(* IEC 61131-3 sources: vertical-injection-machine-docs/docs/IM_SYS_PRG/Code/主程序入口, 8 files *)

(* ---- MachineControlTypes.st ---- *)
(*
  MachineControlTypes.st
  功能：
  1. 定义机器级主控入口使用的命令、参数、传感器和状态结构。
  2. 统一手动、调模、半自动、全自动四类运行方式的上层接口。
  3. 为 `FB_MachineController` 和 `PRG_MainControl` 提供稳定的数据边界。

  说明：
  1. 现有各 `FB_*` 子模块仍然保持模块级职责，不在这里重复定义工艺细节。
  2. 机器级接口只负责把分散的模块输入输出汇总成“可实例化、可调用、可监控”的主控层。
  3. 后续若增加新轴、新模块或新工艺模式，应优先扩展本文件，再扩展主控逻辑。
*)

TYPE ST_MachineManualCommand :
STRUCT
    (* 合模模块手动命令。uiClampMode 沿用模块定义：1/2 自动开合模，3/4 调试开合模。 *)
    bClampStart: BOOL;
    uiClampMode: UINT;

    (* 调模模块手动命令。uiMoldAdjustMode 沿用模块定义：1/2 进退，3/4 手动进退。 *)
    bMoldAdjustStart: BOOL;
    uiMoldAdjustMode: UINT;

    (* 座台模块手动命令。uiNozzleMode 沿用模块定义：1/2 进退，3/4 调试进退。 *)
    bNozzleStart: BOOL;
    uiNozzleMode: UINT;

    (* 射胶模块手动命令。uiInjectMode 沿用模块定义：1/2 射出与射退，3/4 调试。 *)
    bInjectStart: BOOL;
    uiInjectMode: UINT;

    (* 储料模块手动命令。储料块没有独立模式号，手动时只需要启动命令。 *)
    bMeterStart: BOOL;

    (* 托模基础模块手动命令。uiEjectMode 沿用模块定义：1/2 进退，6/7 调试。 *)
    bEjectStart: BOOL;
    uiEjectMode: UINT;

    (* 托模组合模式命令。用于定次、震动、停留等更高层动作。 *)
    bEjectModeStart: BOOL;
    uiEjectPatternMode: UINT;   // 1=定次 2=震动 3=停留
    uiEjectTimes: UINT;         // 定次/震动次数；震动模式下 0 表示持续循环

    (* 中子模块手动命令。uiCoreMode 沿用模块定义：1/2 进退，3/4 调试。 *)
    bCoreStart: BOOL;
    uiCoreMode: UINT;

    (* 温控顶层命令。bTempStart 启动温控；bR0~bR3 可直接下发 4 组加热命令。 *)
    bTempStart: BOOL;          // TRUE=顶层温控块进入执行态。
    bR0: BOOL;                 // TRUE=人工直接驱动第 0 组加热输出。
    bR1: BOOL;                 // TRUE=人工直接驱动第 1 组加热输出。
    bR2: BOOL;                 // TRUE=人工直接驱动第 2 组加热输出。
    bR3: BOOL;                 // TRUE=人工直接驱动第 3 组加热输出。
END_STRUCT
END_TYPE

TYPE ST_MachineCommand :
STRUCT
    (* 机器级公共命令。
       说明：
       1. 该结构既可以作为单一命令源边界，也可以作为顶层仲裁后的最终机器命令边界。
       2. 当前工程先接入面板命令源，再由 `FB_CommandArbiter` 统一生成最终 `gvl_stCommand`。
    *)
    bStart: BOOL;               // 周期启动/当前模块启动
    bStop: BOOL;                // 正常停止
    bEStop: BOOL;               // 急停
    bReset: BOOL;               // 复位所有模块

    (* 运行模式。
       0=停机/待机
       1=手动
       2=半自动
       3=全自动
       4=调模模式

       说明：
       1. 手动模式允许人工点动各模块。
       2. 调模模式是独立机器模式，只开放锁模调试与调模相关动作，
          用于装模、试模和模厚调整，不参与自动循环。
    *)
    uiMachineMode: UINT;

    (* 手动模式与调模模式下的分模块命令集合。
       说明：
       1. 手动模式会读取整套人工命令。
       2. 调模模式只会读取其中与锁模调试、调模和温控相关的命令。
    *)
    stManual: ST_MachineManualCommand;
END_STRUCT
END_TYPE

TYPE ST_MachineModeState :
STRUCT
    (* 机器当前模式解析结果。 *)
    bManualModeActive: BOOL;       // TRUE=当前主控解析出的机器模式为手动模式。
    bMoldAdjustModeActive: BOOL;   // TRUE=当前主控解析出的机器模式为调模模式。
    bSemiAutoModeActive: BOOL;     // TRUE=当前主控解析出的机器模式为半自动模式。
    bFullAutoModeActive: BOOL;     // TRUE=当前主控解析出的机器模式为全自动模式。
    bModeChanged: BOOL;            // TRUE=本拍检测到机器模式发生切换，可用于打一拍总停止保护。
    uiResolvedAutoMode: UINT;      // 自动流程专用模式号；0=非自动 1=半自动 2=全自动。
    bGlobalStop: BOOL;             // 主控统一停止位；收口停机命令、停机模式和切模保护停止。
END_STRUCT
END_TYPE

TYPE ST_MachineModuleCommands :
STRUCT
    (* 合模块最终命令。 *)
    bClampStart: BOOL;             // TRUE=主控最终允许合模块启动当前动作。
    bClampReset: BOOL;             // TRUE=主控最终要求合模块回到复位态。
    uiClampMode: UINT;             // 主控最终下发给合模块的动作模式号。

    (* 调模块最终命令。 *)
    bMoldAdjustStart: BOOL;        // TRUE=主控最终允许调模块启动当前动作。
    bMoldAdjustReset: BOOL;        // TRUE=主控最终要求调模块回到复位态。
    uiMoldAdjustMode: UINT;        // 主控最终下发给调模块的动作模式号。

    (* 座台模块最终命令。 *)
    bNozzleStart: BOOL;            // TRUE=主控最终允许座台模块启动当前动作。
    bNozzleReset: BOOL;            // TRUE=主控最终要求座台模块回到复位态。
    uiNozzleMode: UINT;            // 主控最终下发给座台模块的动作模式号。

    (* 射胶模块最终命令。 *)
    bInjectStart: BOOL;            // TRUE=主控最终允许射胶模块启动当前动作。
    bInjectReset: BOOL;            // TRUE=主控最终要求射胶模块回到复位态。
    uiInjectMode: UINT;            // 主控最终下发给射胶模块的动作模式号。

    (* 储料模块最终命令。 *)
    bMeterStart: BOOL;             // TRUE=主控最终允许储料模块启动当前动作。
    bMeterReset: BOOL;             // TRUE=主控最终要求储料模块回到复位态。

    (* 基础托模块最终命令。 *)
    bEjectStart: BOOL;             // TRUE=主控最终允许基础托模块启动当前动作。
    bEjectReset: BOOL;             // TRUE=主控最终要求基础托模块回到复位态。
    uiEjectMode: UINT;             // 主控最终下发给基础托模块的动作模式号。

    (* 托模组合模式块最终命令。 *)
    bEjectModeStart: BOOL;         // TRUE=主控最终允许托模组合模式块启动当前动作。
    bEjectModeReset: BOOL;         // TRUE=主控最终要求托模组合模式块回到复位态。
    uiEjectPatternMode: UINT;      // 主控最终下发给托模组合模式块的组合模式号。
    uiEjectTimes: UINT;            // 主控最终下发给托模组合模式块的循环次数或震动次数。

    (* 中子模块最终命令。 *)
    bCoreStart: BOOL;              // TRUE=主控最终允许中子模块启动当前动作。
    bCoreReset: BOOL;              // TRUE=主控最终要求中子模块回到复位态。
    uiCoreMode: UINT;              // 主控最终下发给中子模块的动作模式号。
END_STRUCT
END_TYPE

TYPE ST_MachineSensor :
STRUCT
    (* 机器公共条件。自动流程会优先检查这些前提是否满足。 *)
    bDoorClosed: BOOL;
    bHydReady: BOOL;
    bSystemNoAlarm: BOOL;

    (* 合模模块过程信号。 *)
    bOpenStop: BOOL;
    bCloseLowPres: BOOL;
    bCloseHighPres: BOOL;
    bCloseStop: BOOL;
    udiClampElecRulerVal: UDINT;
    uiClampPresElecRulerVal: UINT;

    (* 调模模块过程信号。 *)
    bMoldAdjustInStop: BOOL;
    bMoldAdjustOutStop: BOOL;

    (* 座台模块过程信号。 *)
    bNozzleInStop: BOOL;
    bNozzleOutStop: BOOL;
    udiNozzleElecRulerVal: UDINT;

    (* 射胶与储料模块过程信号。 *)
    bInjSeg1Stop: BOOL;
    bInjSeg2Stop: BOOL;
    bInjStop: BOOL;
    bSuckBackStop: BOOL;
    bMeterStop: BOOL;
    udiInjElecRulerVal: UDINT;

    (* 托模模块过程信号。 *)
    bEjectInStop: BOOL;
    bEjectOutStop: BOOL;
    udiEjectElecRulerVal: UDINT;

    (* 中子模块过程信号。 *)
    bCoreInStop: BOOL;
    bCoreOutStop: BOOL;

    (* 轴反馈。
       这些反馈值会经由子模块接口写回各自的 `ST_AxisRefHyd`，让模块层同时看到“设定值”和“实际值”。
    *)
    rClampActualPosition: LREAL;
    rClampActualVelocity: LREAL;
    rClampActualPressure: LREAL;

    rMoldAdjustActualPosition: LREAL;
    rMoldAdjustActualVelocity: LREAL;
    rMoldAdjustActualPressure: LREAL;

    rNozzleActualPosition: LREAL;
    rNozzleActualVelocity: LREAL;
    rNozzleActualPressure: LREAL;

    rInjectActualPosition: LREAL;
    rInjectActualVelocity: LREAL;
    rInjectActualPressure: LREAL;

    rMeterActualPosition: LREAL;
    rMeterActualVelocity: LREAL;
    rMeterActualPressure: LREAL;

    rEjectActualPosition: LREAL;
    rEjectActualVelocity: LREAL;
    rEjectActualPressure: LREAL;

    rCoreActualPosition: LREAL;
    rCoreActualVelocity: LREAL;
    rCoreActualPressure: LREAL;
END_STRUCT
END_TYPE

TYPE ST_MachinePara :
STRUCT
    (* 子模块工艺参数全集。
       说明：
       1. 这是机器当前在线运行参数。
       2. `FB_MachineController` 只读取并分发，不在内部改写这些工艺值。
       3. 若 HMI 需要统一配方编辑入口，建议通过专用 HMI 参数接口先写入编辑缓冲区，
          再由上层执行“应用到机器”动作，避免画面直接改动在线参数。
    *)
    stClampPara: ST_ClampPara;
    stMoldAdjustPara: ST_MoldAdjustPara;
    stNozzlePara: ST_NozzlePara;
    stInjectPara: ST_InjectPara;
    stMeterPara: ST_MeterPara;
    stEjectPara: ST_EjectPara;
    stCorePara: ST_CorePara;
    stEK312InPara: ST_EK312InPara;
    stAutoPara: ST_AutoCyclePara;
END_STRUCT
END_TYPE

TYPE ST_HMIRecipeMeta :
STRUCT
    (* HMI 配方基础信息。
       这些字段不直接参与动作控制，但便于画面做配方编号、名称、版本和脏数据管理。
    *)
    uiRecipeID: UINT;             // HMI 配方号/工艺号
    sRecipeName: STRING[40];      // HMI 显示用配方名称
    uiRecipeVersion: UINT;        // HMI 自管版本号，可在每次保存后自增
    bDirty: BOOL;                 // TRUE=HMI 编辑缓冲区已改动但还未下发到机器
END_STRUCT
END_TYPE

TYPE ST_HMIProcessPara :
STRUCT
    (* HMI 统一工艺参数接口。
       说明：
       1. HMI 只需要绑定这一套结构，就能覆盖整机全部工艺参数。
       2. 内部仍复用各模块原生参数结构，避免为了画面再拆一层重复字段。
       3. `stMachinePara` 是 HMI 编辑缓冲区，不等同于当前在线运行参数。
          只有执行“应用到机器”后，内容才会写入在线参数。
       4. HMI 画面在用户改动任意字段后，建议同步把 `stMeta.bDirty` 置为 TRUE，
          便于配方页显示“已编辑未下发/未保存”状态。
    *)
    stMeta: ST_HMIRecipeMeta;
    stMachinePara: ST_MachinePara;
END_STRUCT
END_TYPE

TYPE ST_HMIParaCommand :
STRUCT
    (* HMI 参数同步命令。
       这些信号建议由按钮上升沿触发，不建议长时间保持 TRUE。
    *)
    bReadMachinePara: BOOL;       // 把当前在线运行参数读回到 HMI 编辑缓冲区
    bApplyToMachine: BOOL;        // 把 HMI 编辑缓冲区参数应用到机器在线参数
    bClearDirty: BOOL;            // 人工清除 HMI 编辑脏标记
END_STRUCT
END_TYPE

TYPE ST_HMIParaStatus :
STRUCT
    (* HMI 参数接口状态。
       这些状态用于给 HMI 做按钮反馈、提示灯和下发拦截提示。
    *)
    bInitialized: BOOL;           // TRUE=已完成首次把在线参数装载到 HMI 缓冲区
    bMachineParaLocked: BOOL;     // TRUE=机器正在运行/忙碌，禁止下发工艺参数
    bReadDone: BOOL;              // 本扫描周期完成了一次在线参数读回
    bApplyDone: BOOL;             // 本扫描周期完成了一次工艺参数下发
    bClearDone: BOOL;             // 本扫描周期完成了一次脏标记清除
    bApplyBlocked: BOOL;          // 本扫描周期收到下发命令但被拦截
    uiLastAction: UINT;           // 0=无 1=首次装载 2=读取在线参数 3=应用到机器 4=清除脏标记 5=下发被拦截
    uiLastRejectReason: UINT;     // 0=无 1=机器忙碌
    uiSyncCount: UINT;            // 成功同步次数统计
    uiRecipeID: UINT;             // 当前 HMI 缓冲区配方号镜像
    uiRecipeVersion: UINT;        // 当前 HMI 缓冲区版本号镜像
    sRecipeName: STRING[40];      // 当前 HMI 缓冲区名称镜像
    bDirty: BOOL;                 // 当前 HMI 缓冲区脏标记镜像
END_STRUCT
END_TYPE

TYPE ST_MachineStatus :
STRUCT
    (* 机器级总状态。 *)
    uiMachineMode: UINT;
    bManualModeActive: BOOL;
    bMoldAdjustModeActive: BOOL;
    bSemiAutoModeActive: BOOL;
    bFullAutoModeActive: BOOL;
    bAutoReady: BOOL;
    bMachineBusy: BOOL;
    bMachineDone: BOOL;
    bMachineAlarm: BOOL;
    dwMachineAlarmID: DWORD;
    uiMachineActHint: UINT;
    uiMachineActTime: UINT;
    uiCycleCount: UINT;

    (* 自动流程状态。 *)
    bAutoBusy: BOOL;
    bAutoDone: BOOL;
    bAutoAlarm: BOOL;
    dwAutoAlarmID: DWORD;

    (* 合模模块状态。 *)
    bClampBusy: BOOL;
    bClampDone: BOOL;
    bClampAlarm: BOOL;
    dwClampAlarmID: DWORD;
    bMoldOpened: BOOL;
    bMoldClosed: BOOL;

    (* 调模模块状态。 *)
    bMoldAdjustBusy: BOOL;
    bMoldAdjustDone: BOOL;
    bMoldAdjustAlarm: BOOL;
    dwMoldAdjustAlarmID: DWORD;
    bMoldAdjustIned: BOOL;
    bMoldAdjustOuted: BOOL;

    (* 座台模块状态。 *)
    bNozzleBusy: BOOL;
    bNozzleDone: BOOL;
    bNozzleAlarm: BOOL;
    dwNozzleAlarmID: DWORD;
    bNozzleIned: BOOL;
    bNozzleOuted: BOOL;

    (* 射胶模块状态。 *)
    bInjectBusy: BOOL;
    bInjectDone: BOOL;
    bInjectAlarm: BOOL;
    dwInjectAlarmID: DWORD;
    bInjected: BOOL;
    bHeld: BOOL;
    bSuckBacked: BOOL;

    (* 储料模块状态。 *)
    bMeterBusy: BOOL;
    bMeterDone: BOOL;
    bMeterAlarm: BOOL;
    dwMeterAlarmID: DWORD;
    bMetered: BOOL;

    (* 托模模块状态。
       bEjectModeSelected=TRUE 时表示当前输出来自 `FB_EjectMode`；
       否则当前输出来自基础 `FB_Eject`。
    *)
    bEjectModeSelected: BOOL;
    bEjectBusy: BOOL;
    bEjectDone: BOOL;
    bEjectAlarm: BOOL;
    dwEjectAlarmID: DWORD;
    bEjectIned: BOOL;
    bEjectOuted: BOOL;

    (* 中子模块状态。 *)
    bCoreBusy: BOOL;
    bCoreDone: BOOL;
    bCoreAlarm: BOOL;
    dwCoreAlarmID: DWORD;
    bCoreIned: BOOL;
    bCoreOuted: BOOL;

END_STRUCT
END_TYPE

(* ---- FB_CommandArbiter.st ---- *)
(*
  FB_CommandArbiter 功能块
  功能：
  1. 统一收口顶层不同来源的机器命令，再输出给 `FB_MachineController` 与其他顶层消费者。
  2. 当前版本先保留外部入口已经写入的基础公共命令，再用面板命令源覆盖模式与手动字段。
  3. 后续若接入 HMI 运行命令、远程命令或调试命令，应优先在本块扩展优先级与仲裁规则。
*)
FUNCTION_BLOCK FB_CommandArbiter
VAR_INPUT
    stBaseCommandIn: ST_MachineCommand;          // 其他外部入口当前写入的基础机器命令快照；当前版本优先保留其公共启动/停止/复位类字段。
    stPanelCommandSourceIn: ST_MachineCommand;   // 面板调度层输出的机器命令源；当前版本只用本源覆盖模式与手动字段，不直接覆盖公共启动/停止/复位类字段。
END_VAR
VAR_OUTPUT
    stCommandOut: ST_MachineCommand;             // 仲裁后的最终机器命令；供顶层温控和机器主控统一消费。
END_VAR

(* 当前版本的仲裁策略：
   1. 先保留外部基础命令快照中的公共启动/停止/复位/EStop 字段。
   2. 再用面板命令源覆盖它真正负责的模式与手动点动字段。
   3. 这里保留独立功能块，是为了后续增加新命令源时不再修改顶层调用链。
*)
stCommandOut := stBaseCommandIn;                                               // 先复制当前扫描周期的基础机器命令快照，保留外部入口写入的公共控制字段。

IF stPanelCommandSourceIn.uiMachineMode <> UINT#0 THEN
    stCommandOut.uiMachineMode := stPanelCommandSourceIn.uiMachineMode;         // 面板只要给出了有效模式号，就由面板模式选择覆盖当前最终机器模式。
END_IF;

stCommandOut.stManual.bClampStart := stPanelCommandSourceIn.stManual.bClampStart;                 // 合模点动命令由面板源直接覆盖最终手动命令。
stCommandOut.stManual.uiClampMode := stPanelCommandSourceIn.stManual.uiClampMode;                 // 合模点动模式号由面板源直接覆盖最终手动命令。
stCommandOut.stManual.bMoldAdjustStart := stPanelCommandSourceIn.stManual.bMoldAdjustStart;       // 调模点动命令由面板源直接覆盖最终手动命令。
stCommandOut.stManual.uiMoldAdjustMode := stPanelCommandSourceIn.stManual.uiMoldAdjustMode;       // 调模点动模式号由面板源直接覆盖最终手动命令。
stCommandOut.stManual.bNozzleStart := stPanelCommandSourceIn.stManual.bNozzleStart;               // 座台点动命令由面板源直接覆盖最终手动命令。
stCommandOut.stManual.uiNozzleMode := stPanelCommandSourceIn.stManual.uiNozzleMode;               // 座台点动模式号由面板源直接覆盖最终手动命令。
stCommandOut.stManual.bInjectStart := stPanelCommandSourceIn.stManual.bInjectStart;               // 射胶点动命令由面板源直接覆盖最终手动命令。
stCommandOut.stManual.uiInjectMode := stPanelCommandSourceIn.stManual.uiInjectMode;               // 射胶点动模式号由面板源直接覆盖最终手动命令。
stCommandOut.stManual.bMeterStart := stPanelCommandSourceIn.stManual.bMeterStart;                 // 储料点动命令由面板源直接覆盖最终手动命令。
stCommandOut.stManual.bEjectStart := stPanelCommandSourceIn.stManual.bEjectStart;                 // 基础托模点动命令由面板源直接覆盖最终手动命令。
stCommandOut.stManual.uiEjectMode := stPanelCommandSourceIn.stManual.uiEjectMode;                 // 基础托模模式号由面板源直接覆盖最终手动命令。
stCommandOut.stManual.bEjectModeStart := stPanelCommandSourceIn.stManual.bEjectModeStart;         // 托模组合模式启动命令由面板源直接覆盖最终手动命令。
stCommandOut.stManual.uiEjectPatternMode := stPanelCommandSourceIn.stManual.uiEjectPatternMode;   // 托模组合模式号由面板源直接覆盖最终手动命令。
stCommandOut.stManual.uiEjectTimes := stPanelCommandSourceIn.stManual.uiEjectTimes;               // 托模组合次数由面板源直接覆盖最终手动命令。
stCommandOut.stManual.bCoreStart := stPanelCommandSourceIn.stManual.bCoreStart;                   // 中子点动命令由面板源直接覆盖最终手动命令。
stCommandOut.stManual.uiCoreMode := stPanelCommandSourceIn.stManual.uiCoreMode;                   // 中子点动模式号由面板源直接覆盖最终手动命令。
stCommandOut.stManual.bTempStart := stPanelCommandSourceIn.stManual.bTempStart;                   // 温控开关锁存值由面板源直接覆盖最终手动命令。
stCommandOut.stManual.bR0 := stPanelCommandSourceIn.stManual.bR0;                                 // 温控人工组 0 命令由面板源直接覆盖最终手动命令。
stCommandOut.stManual.bR1 := stPanelCommandSourceIn.stManual.bR1;                                 // 温控人工组 1 命令由面板源直接覆盖最终手动命令。
stCommandOut.stManual.bR2 := stPanelCommandSourceIn.stManual.bR2;                                 // 温控人工组 2 命令由面板源直接覆盖最终手动命令。
stCommandOut.stManual.bR3 := stPanelCommandSourceIn.stManual.bR3;                                 // 温控人工组 3 命令由面板源直接覆盖最终手动命令。
END_FUNCTION_BLOCK

(* ---- FB_MachineCommandComposer.st ---- *)
(*
  FB_MachineCommandComposer 功能块
  功能：
  1. 把手动、调模和自动三类来源的模块命令合成为一套最终执行命令。
  2. 把基础托模块与托模组合模式块的互斥选择统一收口，避免双块抢同一根轴。
  3. 当前块只负责命令合成，不直接调用任何执行模块。
*)
FUNCTION_BLOCK FB_MachineCommandComposer
VAR_INPUT
    stCommand: ST_MachineCommand;            // 顶层下发的最终机器命令；当前块只消费公共复位命令与手动命令结构。
    stModeState: ST_MachineModeState;        // 当前扫描周期解析出的模式状态结构；决定最终命令应由哪一类来源接管。

    (* 手动/调模路由结果。 *)
    bManualClampStart: BOOL;                 // 手动或调模路由给出的合模启动命令。
    uiManualClampMode: UINT;                 // 手动或调模路由给出的合模模式号。
    bManualMoldAdjustStart: BOOL;            // 手动或调模路由给出的调模启动命令。
    uiManualMoldAdjustMode: UINT;            // 手动或调模路由给出的调模模式号。
    bManualNozzleStart: BOOL;                // 手动路由给出的座台启动命令。
    uiManualNozzleMode: UINT;                // 手动路由给出的座台模式号。
    bManualInjectStart: BOOL;                // 手动路由给出的射胶启动命令。
    uiManualInjectMode: UINT;                // 手动路由给出的射胶模式号。
    bManualMeterStart: BOOL;                 // 手动路由给出的储料启动命令。
    bManualEjectStart: BOOL;                 // 手动路由给出的基础托模启动命令。
    uiManualEjectMode: UINT;                 // 手动路由给出的基础托模模式号。
    bManualEjectModeStart: BOOL;             // 手动路由给出的托模组合模式启动命令。
    uiManualEjectPatternMode: UINT;          // 手动路由给出的托模组合模式号。
    uiManualEjectTimes: UINT;                // 手动路由给出的托模组合次数或震动次数。
    bManualCoreStart: BOOL;                  // 手动路由给出的中子启动命令。
    uiManualCoreMode: UINT;                  // 手动路由给出的中子模式号。

    (* 自动流程输出结果。 *)
    bAutoClampStart: BOOL;                   // 自动流程给出的合模启动命令。
    bAutoClampReset: BOOL;                   // 自动流程给出的合模复位命令。
    uiAutoClampMode: UINT;                   // 自动流程给出的合模模式号。
    bAutoNozzleStart: BOOL;                  // 自动流程给出的座台启动命令。
    bAutoNozzleReset: BOOL;                  // 自动流程给出的座台复位命令。
    uiAutoNozzleMode: UINT;                  // 自动流程给出的座台模式号。
    bAutoInjectStart: BOOL;                  // 自动流程给出的射胶启动命令。
    bAutoInjectReset: BOOL;                  // 自动流程给出的射胶复位命令。
    uiAutoInjectMode: UINT;                  // 自动流程给出的射胶模式号。
    bAutoMeterStart: BOOL;                   // 自动流程给出的储料启动命令。
    bAutoMeterReset: BOOL;                   // 自动流程给出的储料复位命令。
    bAutoEjectStart: BOOL;                   // 自动流程给出的基础托模启动命令。
    bAutoEjectReset: BOOL;                   // 自动流程给出的基础托模复位命令。
    uiAutoEjectMode: UINT;                   // 自动流程给出的基础托模模式号。
END_VAR
VAR_OUTPUT
    stModuleCommands: ST_MachineModuleCommands; // 主控最终下发给各执行模块的统一命令集合。
    bUseEjectModeManual: BOOL;                  // TRUE=当前应切换到托模组合模式块，而不是基础托模块。
END_VAR

(* 先给各模块命令做安全缺省值。
   这样在模式切换时，未被当前模式接管的模块会自然保持停止/复位，不会沿用旧命令。
*)
stModuleCommands.bClampStart := FALSE;                          // 默认不给合模块启动命令，避免未被接管时沿用旧动作。
stModuleCommands.bClampReset := stCommand.bReset;              // 合模块默认只响应顶层复位命令。
stModuleCommands.uiClampMode := 0;                             // 合模块默认模式号清零，表示当前无有效动作。

stModuleCommands.bMoldAdjustStart := FALSE;                    // 默认不给调模块启动命令，避免未被接管时沿用旧动作。
stModuleCommands.bMoldAdjustReset := stCommand.bReset;         // 调模块默认只响应顶层复位命令。
stModuleCommands.uiMoldAdjustMode := 0;                        // 调模块默认模式号清零，表示当前无有效动作。

stModuleCommands.bNozzleStart := FALSE;                        // 默认不给座台模块启动命令，避免未被接管时沿用旧动作。
stModuleCommands.bNozzleReset := stCommand.bReset;             // 座台模块默认只响应顶层复位命令。
stModuleCommands.uiNozzleMode := 0;                            // 座台模块默认模式号清零，表示当前无有效动作。

stModuleCommands.bInjectStart := FALSE;                        // 默认不给射胶模块启动命令，避免未被接管时沿用旧动作。
stModuleCommands.bInjectReset := stCommand.bReset;             // 射胶模块默认只响应顶层复位命令。
stModuleCommands.uiInjectMode := 0;                            // 射胶模块默认模式号清零，表示当前无有效动作。

stModuleCommands.bMeterStart := FALSE;                         // 默认不给储料模块启动命令，避免未被接管时沿用旧动作。
stModuleCommands.bMeterReset := stCommand.bReset;              // 储料模块默认只响应顶层复位命令。

stModuleCommands.bEjectStart := FALSE;                         // 默认不给基础托模块启动命令，避免未被接管时沿用旧动作。
stModuleCommands.bEjectReset := stCommand.bReset;              // 基础托模块默认只响应顶层复位命令。
stModuleCommands.uiEjectMode := 0;                             // 基础托模块默认模式号清零，表示当前无有效动作。

stModuleCommands.bEjectModeStart := FALSE;                     // 默认不给托模模式块启动命令，避免组合模式在切模后残留。
stModuleCommands.bEjectModeReset := TRUE;                      // 默认把托模模式块拉在复位态，只有明确使用时才释放。
stModuleCommands.uiEjectPatternMode := 0;                      // 托模模式块默认模式号清零，表示当前不执行组合动作。
stModuleCommands.uiEjectTimes := 0;                            // 托模模式块默认次数清零，避免沿用上一轮次数设定。

stModuleCommands.bCoreStart := FALSE;                          // 默认不给中子模块启动命令，避免未被接管时沿用旧动作。
stModuleCommands.bCoreReset := stCommand.bReset;               // 中子模块默认只响应顶层复位命令。
stModuleCommands.uiCoreMode := 0;                              // 中子模块默认模式号清零，表示当前无有效动作。

(* 把不同来源的命令合并为“最终执行命令”。
   1. 手动模式：手动命令由 `FB_ManualMode` 路由。
   2. 调模模式：命令由 `FB_MoldAdjustMode` 路由，锁模强制进入调试方向，其他模块保持停机。
   3. 自动模式：命令来自 `FB_AutoCycle` 的调度输出。
*)
IF stModeState.bManualModeActive THEN
    stModuleCommands.bClampStart := bManualClampStart;             // 手动模式下，合模块直接接收手动命令路由结果。
    stModuleCommands.uiClampMode := uiManualClampMode;             // 手动模式下，合模块直接接收手动动作模式号。

    stModuleCommands.bMoldAdjustStart := bManualMoldAdjustStart;   // 手动模式下，调模块直接接收手动命令路由结果。
    stModuleCommands.uiMoldAdjustMode := uiManualMoldAdjustMode;   // 手动模式下，调模块直接接收手动动作模式号。

    stModuleCommands.bNozzleStart := bManualNozzleStart;           // 手动模式下，座台模块直接接收手动命令路由结果。
    stModuleCommands.uiNozzleMode := uiManualNozzleMode;           // 手动模式下，座台模块直接接收手动动作模式号。

    stModuleCommands.bInjectStart := bManualInjectStart;           // 手动模式下，射胶模块直接接收手动命令路由结果。
    stModuleCommands.uiInjectMode := uiManualInjectMode;           // 手动模式下，射胶模块直接接收手动动作模式号。

    stModuleCommands.bMeterStart := bManualMeterStart;             // 手动模式下，储料模块直接接收手动启动命令。

    stModuleCommands.bCoreStart := bManualCoreStart;               // 手动模式下，中子模块直接接收手动命令路由结果。
    stModuleCommands.uiCoreMode := uiManualCoreMode;               // 手动模式下，中子模块直接接收手动动作模式号。
ELSIF stModeState.bMoldAdjustModeActive THEN
    stModuleCommands.bClampStart := bManualClampStart;             // 调模模式下，锁模动作仍由调模命令路由结果接管。
    stModuleCommands.uiClampMode := uiManualClampMode;             // 调模模式下，锁模模式号仍取自调模命令路由结果。

    stModuleCommands.bMoldAdjustStart := bManualMoldAdjustStart;   // 调模模式下，调模块直接接收调模命令路由结果。
    stModuleCommands.uiMoldAdjustMode := uiManualMoldAdjustMode;   // 调模模式下，调模块直接接收调模动作模式号。
ELSE
    stModuleCommands.bClampStart := bAutoClampStart;               // 自动模式下，合模块启动命令由自动流程输出接管。
    stModuleCommands.bClampReset := stCommand.bReset OR bAutoClampReset; // 自动模式下，顶层复位与自动步骤复位任一成立都可复位合模块。
    stModuleCommands.uiClampMode := uiAutoClampMode;               // 自动模式下，合模块动作模式号由自动流程给定。

    stModuleCommands.bNozzleStart := bAutoNozzleStart;             // 自动模式下，座台模块启动命令由自动流程输出接管。
    stModuleCommands.bNozzleReset := stCommand.bReset OR bAutoNozzleReset; // 自动模式下，顶层复位与自动步骤复位任一成立都可复位座台模块。
    stModuleCommands.uiNozzleMode := uiAutoNozzleMode;             // 自动模式下，座台模块动作模式号由自动流程给定。

    stModuleCommands.bInjectStart := bAutoInjectStart;             // 自动模式下，射胶模块启动命令由自动流程输出接管。
    stModuleCommands.bInjectReset := stCommand.bReset OR bAutoInjectReset; // 自动模式下，顶层复位与自动步骤复位任一成立都可复位射胶模块。
    stModuleCommands.uiInjectMode := uiAutoInjectMode;             // 自动模式下，射胶模块动作模式号由自动流程给定。

    stModuleCommands.bMeterStart := bAutoMeterStart;               // 自动模式下，储料模块启动命令由自动流程输出接管。
    stModuleCommands.bMeterReset := stCommand.bReset OR bAutoMeterReset; // 自动模式下，顶层复位与自动步骤复位任一成立都可复位储料模块。

    stModuleCommands.bEjectStart := bAutoEjectStart;               // 自动模式下，基础托模块启动命令由自动流程输出接管。
    stModuleCommands.bEjectReset := stCommand.bReset OR bAutoEjectReset; // 自动模式下，顶层复位与自动步骤复位任一成立都可复位基础托模块。
    stModuleCommands.uiEjectMode := uiAutoEjectMode;               // 自动模式下，基础托模块动作模式号由自动流程给定。
END_IF;

(* 托模既有基础动作块，也有组合模式块。
   这里把两类命令拆开，避免两个功能块同时争抢同一输出轴。
*)
bUseEjectModeManual := stModeState.bManualModeActive AND bManualEjectModeStart AND   // 只有手动模式下明确发起托模模式命令时，才允许切到组合托模块。
    (uiManualEjectPatternMode >= 1) AND                                               // 模式号下限必须落在当前支持的托模组合模式范围内。
    (uiManualEjectPatternMode <= 3);                                                  // 模式号上限必须落在当前支持的托模组合模式范围内。

IF stModeState.bManualModeActive AND (NOT bUseEjectModeManual) THEN
    stModuleCommands.bEjectStart := bManualEjectStart;               // 纯手动基础托模时，把基础托模启动命令路由给 `FB_Eject`。
    stModuleCommands.bEjectReset := stCommand.bReset;                // 纯手动基础托模时，基础托模块只响应顶层复位命令。
    stModuleCommands.uiEjectMode := uiManualEjectMode;               // 纯手动基础托模时，把手动托模模式号路由给 `FB_Eject`。
ELSIF NOT stModeState.bManualModeActive THEN
    stModuleCommands.bEjectStart := bAutoEjectStart;                 // 非手动模式下，基础托模块启动命令由自动流程输出接管。
    stModuleCommands.bEjectReset := stCommand.bReset OR bAutoEjectReset; // 非手动模式下，顶层复位与自动步骤复位任一成立都可复位基础托模块。
    stModuleCommands.uiEjectMode := uiAutoEjectMode;                 // 非手动模式下，基础托模块动作模式号由自动流程给定。
ELSE
    stModuleCommands.bEjectStart := FALSE;                           // 进入托模组合模式时，强制撤销基础托模块启动命令，避免双块抢轴。
    stModuleCommands.bEjectReset := TRUE;                            // 进入托模组合模式时，强制把基础托模块拉回复位态。
    stModuleCommands.uiEjectMode := 0;                               // 进入托模组合模式时，基础托模块模式号清零。
END_IF;

IF bUseEjectModeManual THEN
    stModuleCommands.bEjectModeStart := bManualEjectModeStart;       // 仅在手动组合托模生效时，把启动命令路由给 `FB_EjectMode`。
    stModuleCommands.bEjectModeReset := stCommand.bReset;            // 仅在手动组合托模生效时，把顶层复位命令路由给 `FB_EjectMode`。
    stModuleCommands.uiEjectPatternMode := uiManualEjectPatternMode; // 仅在手动组合托模生效时，把托模组合模式号路由给 `FB_EjectMode`。
    stModuleCommands.uiEjectTimes := uiManualEjectTimes;             // 仅在手动组合托模生效时，把循环次数或震动次数路由给 `FB_EjectMode`。
END_IF;
END_FUNCTION_BLOCK

(* ---- FB_MachineController.st ---- *)
(*
  FB_MachineController 功能块
  功能：
  1. 提供真正的机器级执行层，负责实例化并周期调用所有模块级功能块。
  2. 通过内部辅助层完成模式解析、命令合成，并把最终模块命令分发给各执行块。
  3. 把模块状态、轴命令和自动流程状态汇总为统一的机器级状态输出。

  调用关系：
  1. `FB_MachineModeResolver` 只负责模式解析，不直接驱动任何执行模块。
  2. `FB_AutoCycle` 只负责调度，不直接驱动任何轴；`FB_MachineCommandComposer` 负责把自动、手动和调模命令收口为最终模块命令。
  3. 各执行模块内部各自持有 `FB_HydAxis` 并自行处理轴使能、轴配置和轴状态并入。
  4. `FB_MachineStatusAggregator` 负责把自动流程和模块状态收口为机器总状态。
  5. `FB_EK312` 由 `PROGRAM PRG_MainControl` 顶层独立调用，本功能块不处理温控块接口和温控状态。
  6. 必须由 `PROGRAM PRG_MainControl` 以 1ms 基础任务调用本功能块；10ms 工艺节拍也必须由顶层生成后通过输入接口送入本块。
*)
FUNCTION_BLOCK FB_MachineController
VAR_INPUT
    stCommand: ST_MachineCommand;    // 顶层下发的机器公共命令集合，包含启动/停止/复位/模式号以及手动动作命令。
    stPara: ST_MachinePara;          // 顶层下发的机器在线工艺参数全集，由主控分发给各执行模块使用。
    stSensor: ST_MachineSensor;      // 顶层采集的现场条件、限位和轴反馈，供主控与子模块做互锁和状态判断。
    bLogicTick10msIn: BOOL;          // 顶层当前扫描周期给出的 10ms 工艺逻辑节拍，本块只在该拍刷新模式路由和自动流程。
END_VAR
VAR_OUTPUT
    stStatus: ST_MachineStatus;      // 主控汇总后的机器级总状态，供 HMI、上位机和其他顶层逻辑统一读取。

    (* 各轴输出。
       这些结构体同时包含模块下发的设定值与主控层回写的实际反馈值，
       便于后续继续接入真实轴控或液压阀控层。
    *)
    stClampAxis: ST_AxisRefHyd;          // 合模模块输出的最终轴命令与反馈镜像，对外暴露为锁模轴边界。
    stMoldAdjustAxis: ST_AxisRefHyd;     // 调模模块输出的最终轴命令与反馈镜像，对外暴露为调模轴边界。
    stNozzleAxis: ST_AxisRefHyd;         // 座台模块输出的最终轴命令与反馈镜像，对外暴露为座台轴边界。
    stInjectAxis: ST_AxisRefHyd;         // 射胶模块输出的最终轴命令与反馈镜像，对外暴露为射胶轴边界。
    stMeterAxis: ST_AxisRefHyd;          // 储料模块输出的最终轴命令与反馈镜像，对外暴露为储料轴边界。
    stEjectAxis: ST_AxisRefHyd;          // 托模模块当前被选中的最终轴命令与反馈镜像，可能来自基础托模或托模模式。
    stCoreAxis: ST_AxisRefHyd;           // 中子模块输出的最终轴命令与反馈镜像，对外暴露为中子轴边界。

    (* 透传关键组合输出。 *)
    aCoreAllow: ARRAY[1..8] OF BOOL;     // 合模模块回写的 8 路中子允许位，供其他模块和上位系统读取联锁结果。
END_VAR
VAR
    (* 子模块实例。 *)
    fbManualMode: FB_ManualMode;                  // 手动模式命令路由实例，把手动按钮翻译成各执行模块可直接消费的命令。
    fbAutoCycle: FB_AutoCycle;                    // 自动流程调度实例，只负责自动步骤编排，不直接操作任何轴。
    fbMoldAdjustMode: FB_MoldAdjustMode;          // 调模模式命令路由实例，把调模专用命令收口到锁模和调模块。
    fbClamp: FB_Clamp;                            // 合模执行模块实例，内部自带锁模轴层处理。
    fbMoldAdjust: FB_MoldAdjust;                  // 调模执行模块实例，内部自带调模轴层处理。
    fbNozzle: FB_Nozzle;                          // 座台执行模块实例，内部自带座台轴层处理。
    fbInject: FB_Inject;                          // 射胶执行模块实例，内部自带射胶轴层处理。
    fbMeter: FB_Meter;                            // 储料执行模块实例，内部自带储料轴层处理。
    fbEject: FB_Eject;                            // 基础托模执行模块实例，内部自带基础托模轴层处理。
    fbEjectMode: FB_EjectMode;                    // 托模模式执行模块实例，内部复用 `FB_Eject` 做组合动作封装。
    fbCore: FB_Core;                              // 中子执行模块实例，内部自带中子轴层处理。

    bManualClampStart: BOOL := FALSE;             // 手动模式输出的合模启动命令缓存，10ms 节拍刷新后再路由到合模块。
    uiManualClampMode: UINT := 0;                 // 手动模式输出的合模动作模式号缓存。
    bManualMoldAdjustStart: BOOL := FALSE;        // 手动/调模模式输出的调模启动命令缓存。
    uiManualMoldAdjustMode: UINT := 0;            // 手动/调模模式输出的调模动作模式号缓存。
    bManualNozzleStart: BOOL := FALSE;            // 手动模式输出的座台启动命令缓存。
    uiManualNozzleMode: UINT := 0;                // 手动模式输出的座台动作模式号缓存。
    bManualInjectStart: BOOL := FALSE;            // 手动模式输出的射胶启动命令缓存。
    uiManualInjectMode: UINT := 0;                // 手动模式输出的射胶动作模式号缓存。
    bManualMeterStart: BOOL := FALSE;             // 手动模式输出的储料启动命令缓存。
    bManualEjectStart: BOOL := FALSE;             // 手动模式输出的基础托模启动命令缓存。
    uiManualEjectMode: UINT := 0;                 // 手动模式输出的基础托模动作模式号缓存。
    bManualEjectModeStart: BOOL := FALSE;         // 手动模式输出的托模组合模式启动命令缓存。
    uiManualEjectPatternMode: UINT := 0;          // 手动模式输出的托模组合模式号缓存，例如定次/震动/停留。
    uiManualEjectTimes: UINT := 0;                // 手动模式输出的托模组合次数缓存，供定次或震动模式使用。
    bManualCoreStart: BOOL := FALSE;              // 手动模式输出的中子启动命令缓存。
    uiManualCoreMode: UINT := 0;                  // 手动模式输出的中子动作模式号缓存。

    (* 托模基础块和托模模式块不能同时写同一根轴。
       因此各自使用独立的内部轴缓存，最后由主控层按模式择一输出到 stEjectAxis。
    *)
    stEjectAxisBase: ST_AxisRefHyd;               // 基础托模块独占使用的托模轴缓存，避免与托模模式块直接争抢同一输出结构。
    stEjectAxisMode: ST_AxisRefHyd;               // 托模模式块独占使用的托模轴缓存，最终再由主控择一输出到 `stEjectAxis`。

    (* 主控辅助分层实例与结构。 *)
    fbModeResolver: FB_MachineModeResolver;       // 模式解析辅助实例；负责解析机器模式、切模状态和统一停止位。
    fbCommandComposer: FB_MachineCommandComposer; // 命令合成辅助实例；负责把手动、调模和自动命令收口为最终模块命令。
    fbStatusAggregator: FB_MachineStatusAggregator; // 状态汇总辅助实例；负责把自动流程与模块状态收口为机器总状态。
    stModeState: ST_MachineModeState;             // 当前扫描周期解析出的模式状态结构；供主控内部统一消费。
    stModuleCommands: ST_MachineModuleCommands;   // 当前扫描周期合成出的最终模块命令集合；供执行模块统一消费。
    bUseEjectModeManual: BOOL := FALSE;           // TRUE=当前手动命令应切换到托模组合模式而不是基础托模块。

    (* 自动流程输出命令缓存。 *)
    bAutoBusy: BOOL := FALSE;                     // 自动流程 Busy 状态缓存，用于机器级状态汇总。
    bAutoDone: BOOL := FALSE;                     // 自动流程 Done 状态缓存，用于机器级状态汇总。
    bAutoAlarm: BOOL := FALSE;                    // 自动流程 Alarm 状态缓存，用于机器级状态汇总。
    dwAutoAlarmID: DWORD := 0;                    // 自动流程报警码缓存。
    uiAutoActHint: UINT := 0;                     // 自动流程动作提示号缓存，用于优先显示机器当前自动步骤。
    uiAutoActTime: UINT := 0;                     // 自动流程当前动作持续时间缓存。
    uiAutoCycleCount: UINT := 0;                  // 自动流程累计循环次数缓存。
    bAutoClampStart: BOOL := FALSE;               // 自动流程输出的合模启动命令缓存。
    bAutoClampReset: BOOL := FALSE;               // 自动流程输出的合模复位命令缓存。
    uiAutoClampMode: UINT := 0;                   // 自动流程输出的合模动作模式号缓存。
    bAutoNozzleStart: BOOL := FALSE;              // 自动流程输出的座台启动命令缓存。
    bAutoNozzleReset: BOOL := FALSE;              // 自动流程输出的座台复位命令缓存。
    uiAutoNozzleMode: UINT := 0;                  // 自动流程输出的座台动作模式号缓存。
    bAutoInjectStart: BOOL := FALSE;              // 自动流程输出的射胶启动命令缓存。
    bAutoInjectReset: BOOL := FALSE;              // 自动流程输出的射胶复位命令缓存。
    uiAutoInjectMode: UINT := 0;                  // 自动流程输出的射胶动作模式号缓存。
    bAutoMeterStart: BOOL := FALSE;               // 自动流程输出的储料启动命令缓存。
    bAutoMeterReset: BOOL := FALSE;               // 自动流程输出的储料复位命令缓存。
    bAutoEjectStart: BOOL := FALSE;               // 自动流程输出的托模启动命令缓存。
    bAutoEjectReset: BOOL := FALSE;               // 自动流程输出的托模复位命令缓存。
    uiAutoEjectMode: UINT := 0;                   // 自动流程输出的托模动作模式号缓存。

    (* 子模块状态缓存。 *)
    bClampBusy: BOOL := FALSE;                    // 合模块 Busy 状态缓存。
    bClampDone: BOOL := FALSE;                    // 合模块 Done 状态缓存。
    bClampAlarm: BOOL := FALSE;                   // 合模块 Alarm 状态缓存。
    dwClampAlarmID: DWORD := 0;                   // 合模块报警码缓存。
    uiClampActHint: UINT := 0;                    // 合模块动作提示号缓存。
    uiClampActTime: UINT := 0;                    // 合模块当前动作持续时间缓存。
    bMoldOpened: BOOL := FALSE;                   // 合模块“已开模到位”状态缓存。
    bMoldClosed: BOOL := FALSE;                   // 合模块“已合模到位”状态缓存。
    aCoreAllowLocal: ARRAY[1..8] OF BOOL;         // 合模块内部给出的 8 路中子允许位缓存，稍后透传到输出数组。

    bMoldAdjustBusy: BOOL := FALSE;               // 调模块 Busy 状态缓存。
    bMoldAdjustDone: BOOL := FALSE;               // 调模块 Done 状态缓存。
    bMoldAdjustAlarm: BOOL := FALSE;              // 调模块 Alarm 状态缓存。
    dwMoldAdjustAlarmID: DWORD := 0;              // 调模块报警码缓存。
    uiMoldAdjustActHint: UINT := 0;               // 调模块动作提示号缓存。
    uiMoldAdjustActTime: UINT := 0;               // 调模块当前动作持续时间缓存。
    bMoldAdjustIned: BOOL := FALSE;               // 调模块“调模进到位”状态缓存。
    bMoldAdjustOuted: BOOL := FALSE;              // 调模块“调模退到位”状态缓存。

    bNozzleBusy: BOOL := FALSE;                   // 座台模块 Busy 状态缓存。
    bNozzleDone: BOOL := FALSE;                   // 座台模块 Done 状态缓存。
    bNozzleAlarm: BOOL := FALSE;                  // 座台模块 Alarm 状态缓存。
    dwNozzleAlarmID: DWORD := 0;                  // 座台模块报警码缓存。
    uiNozzleActHint: UINT := 0;                   // 座台模块动作提示号缓存。
    uiNozzleActTime: UINT := 0;                   // 座台模块当前动作持续时间缓存。
    bNozzleIned: BOOL := FALSE;                   // 座台模块“进到位”状态缓存。
    bNozzleOuted: BOOL := FALSE;                  // 座台模块“退到位”状态缓存。

    bInjectBusy: BOOL := FALSE;                   // 射胶模块 Busy 状态缓存。
    bInjectDone: BOOL := FALSE;                   // 射胶模块 Done 状态缓存。
    bInjectAlarm: BOOL := FALSE;                  // 射胶模块 Alarm 状态缓存。
    dwInjectAlarmID: DWORD := 0;                  // 射胶模块报警码缓存。
    uiInjectActHint: UINT := 0;                   // 射胶模块动作提示号缓存。
    uiInjectActTime: UINT := 0;                   // 射胶模块当前动作持续时间缓存。
    bInjected: BOOL := FALSE;                     // 射胶模块“射出完成”状态缓存。
    bHeld: BOOL := FALSE;                         // 射胶模块“保压完成”状态缓存。
    bSuckBacked: BOOL := FALSE;                   // 射胶模块“射退完成”状态缓存。

    bMeterBusy: BOOL := FALSE;                    // 储料模块 Busy 状态缓存。
    bMeterDone: BOOL := FALSE;                    // 储料模块 Done 状态缓存。
    bMeterAlarm: BOOL := FALSE;                   // 储料模块 Alarm 状态缓存。
    dwMeterAlarmID: DWORD := 0;                   // 储料模块报警码缓存。
    uiMeterActHint: UINT := 0;                    // 储料模块动作提示号缓存。
    uiMeterActTime: UINT := 0;                    // 储料模块当前动作持续时间缓存。
    bMetered: BOOL := FALSE;                      // 储料模块“储料完成”状态缓存。

    bEjectBaseBusy: BOOL := FALSE;                // 基础托模块 Busy 状态缓存。
    bEjectBaseDone: BOOL := FALSE;                // 基础托模块 Done 状态缓存。
    bEjectBaseAlarm: BOOL := FALSE;               // 基础托模块 Alarm 状态缓存。
    dwEjectBaseAlarmID: DWORD := 0;               // 基础托模块报警码缓存。
    uiEjectBaseActHint: UINT := 0;                // 基础托模块动作提示号缓存。
    uiEjectBaseActTime: UINT := 0;                // 基础托模块当前动作持续时间缓存。
    bEjectBaseIned: BOOL := FALSE;                // 基础托模块“退回到位/内位到位”状态缓存。
    bEjectBaseOuted: BOOL := FALSE;               // 基础托模块“顶出到位/外位到位”状态缓存。

    bEjectModeBusy: BOOL := FALSE;                // 托模模式块 Busy 状态缓存。
    bEjectModeDone: BOOL := FALSE;                // 托模模式块 Done 状态缓存。
    bEjectModeAlarm: BOOL := FALSE;               // 托模模式块 Alarm 状态缓存。
    dwEjectModeAlarmID: DWORD := 0;               // 托模模式块报警码缓存。
    uiEjectModeActHint: UINT := 0;                // 托模模式块动作提示号缓存。
    uiEjectModeActTime: UINT := 0;                // 托模模式块当前动作持续时间缓存。
    bEjectModeIned: BOOL := FALSE;                // 托模模式块“退回到位/内位到位”状态缓存。
    bEjectModeOuted: BOOL := FALSE;               // 托模模式块“顶出到位/外位到位”状态缓存。

    bSelectedEjectBusy: BOOL := FALSE;            // 当前被主控选中的托模来源 Busy 状态缓存。
    bSelectedEjectDone: BOOL := FALSE;            // 当前被主控选中的托模来源 Done 状态缓存。
    bSelectedEjectAlarm: BOOL := FALSE;           // 当前被主控选中的托模来源 Alarm 状态缓存。
    dwSelectedEjectAlarmID: DWORD := 0;           // 当前被主控选中的托模来源报警码缓存。
    uiSelectedEjectActHint: UINT := 0;            // 当前被主控选中的托模来源动作提示号缓存。
    uiSelectedEjectActTime: UINT := 0;            // 当前被主控选中的托模来源动作持续时间缓存。
    bSelectedEjectIned: BOOL := FALSE;            // 当前被主控选中的托模来源“内位到位”状态缓存。
    bSelectedEjectOuted: BOOL := FALSE;           // 当前被主控选中的托模来源“外位到位”状态缓存。

    bCoreBusy: BOOL := FALSE;                     // 中子模块 Busy 状态缓存。
    bCoreDone: BOOL := FALSE;                     // 中子模块 Done 状态缓存。
    bCoreAlarm: BOOL := FALSE;                    // 中子模块 Alarm 状态缓存。
    dwCoreAlarmID: DWORD := 0;                    // 中子模块报警码缓存。
    uiCoreActHint: UINT := 0;                     // 中子模块动作提示号缓存。
    uiCoreActTime: UINT := 0;                     // 中子模块当前动作持续时间缓存。
    bCoreIned: BOOL := FALSE;                     // 中子模块“进到位”状态缓存。
    bCoreOuted: BOOL := FALSE;                    // 中子模块“退到位”状态缓存。

    uiIndex: UINT := 0;                           // 通用数组循环索引，当前用于拷贝 `aCoreAllowLocal` 到输出数组。
END_VAR

(* 运行模式先统一解析，后续所有模块都只看这一组结果。
   其中“调模模式”是机器级独立模式，不等同于普通手动模式：
   1. 只开放锁模调试与调模动作。
   2. 不参与自动循环。
   3. 其他模块保持停机或复位状态，避免试模阶段误动作。
*)
fbModeResolver(
    stCommand := stCommand,                 // 把最终机器命令送入模式解析层，统一生成当前扫描周期的模式状态结构。
    stModeState => stModeState              // 回收本拍解析出的模式状态结构，供后续自动流程、命令合成和状态汇总使用。
);

IF bLogicTick10msIn THEN                                                      // 手动路由、调模路由和自动流程只在顶层送来的 10ms 逻辑拍到来时刷新一次。
    fbManualMode(
        bStop := stModeState.bGlobalStop,                                     // 把主控统一停止位送给手动路由块，切模或停机时立即撤销手动动作。
        bEStop := stCommand.bEStop,                                           // 把急停信号送给手动路由块，确保急停时手动命令立刻失效。
        bReset := stCommand.bReset,                                           // 把顶层复位信号送给手动路由块，便于清空手动命令状态。
        bActive := stModeState.bManualModeActive,                             // 只有机器处于手动模式时，手动路由块才输出有效动作命令。
        stManual := stCommand.stManual,                                       // 把完整手动命令结构送给手动路由块解析。
        bClampStart => bManualClampStart,                                     // 回收手动路由块给出的合模启动命令。
        uiClampMode => uiManualClampMode,                                     // 回收手动路由块给出的合模模式号。
        bMoldAdjustStart => bManualMoldAdjustStart,                           // 回收手动路由块给出的调模启动命令。
        uiMoldAdjustMode => uiManualMoldAdjustMode,                           // 回收手动路由块给出的调模模式号。
        bNozzleStart => bManualNozzleStart,                                   // 回收手动路由块给出的座台启动命令。
        uiNozzleMode => uiManualNozzleMode,                                   // 回收手动路由块给出的座台模式号。
        bInjectStart => bManualInjectStart,                                   // 回收手动路由块给出的射胶启动命令。
        uiInjectMode => uiManualInjectMode,                                   // 回收手动路由块给出的射胶模式号。
        bMeterStart => bManualMeterStart,                                     // 回收手动路由块给出的储料启动命令。
        bEjectStart => bManualEjectStart,                                     // 回收手动路由块给出的基础托模启动命令。
        uiEjectMode => uiManualEjectMode,                                     // 回收手动路由块给出的基础托模模式号。
        bEjectModeStart => bManualEjectModeStart,                             // 回收手动路由块给出的托模组合模式启动命令。
        uiEjectPatternMode => uiManualEjectPatternMode,                       // 回收手动路由块给出的托模组合模式号。
        uiEjectTimes => uiManualEjectTimes,                                   // 回收手动路由块给出的托模组合次数。
        bCoreStart => bManualCoreStart,                                       // 回收手动路由块给出的中子启动命令。
        uiCoreMode => uiManualCoreMode                                        // 回收手动路由块给出的中子模式号。
    );

    fbMoldAdjustMode(
        bStop := stModeState.bGlobalStop,                                     // 把主控统一停止位送给调模路由块，切模或停机时立即撤销调模动作。
        bEStop := stCommand.bEStop,                                           // 把急停信号送给调模路由块，确保急停时调模命令立刻失效。
        bReset := stCommand.bReset,                                           // 把顶层复位信号送给调模路由块，便于清空调模命令状态。
        bActive := stModeState.bMoldAdjustModeActive,                         // 只有机器处于调模模式时，调模路由块才输出有效动作命令。
        stManual := stCommand.stManual,                                       // 把完整手动/调模命令结构送给调模路由块解析。
        bClampStart => bManualClampStart,                                     // 回收调模路由块给出的锁模启动命令。
        uiClampMode => uiManualClampMode,                                     // 回收调模路由块给出的锁模模式号。
        bMoldAdjustStart => bManualMoldAdjustStart,                           // 回收调模路由块给出的调模启动命令。
        uiMoldAdjustMode => uiManualMoldAdjustMode                            // 回收调模路由块给出的调模模式号。
    );
END_IF;

IF bLogicTick10msIn THEN                                                      // 自动流程也只在顶层送来的 10ms 逻辑拍到来时刷新一次。
    (* 自动流程只在半自动/全自动模式下参与调度。
       一旦退出自动模式，就用 bStop 把自动流程拉回空闲态。
    *)
    fbAutoCycle(
        bStart := stCommand.bStart AND (stModeState.uiResolvedAutoMode > 0),
        bStop := stCommand.bStop OR (stModeState.uiResolvedAutoMode = 0),
        bEStop := stCommand.bEStop,
        bReset := stCommand.bReset,
        uiAutoMode := stModeState.uiResolvedAutoMode,
        stAutoPara := stPara.stAutoPara,
        bDoorClosed := stSensor.bDoorClosed,
        bHydReady := stSensor.bHydReady,
        bSystemNoAlarm := stSensor.bSystemNoAlarm AND (NOT bClampAlarm) AND (NOT bMoldAdjustAlarm) AND
            (NOT bNozzleAlarm) AND (NOT bInjectAlarm) AND (NOT bMeterAlarm) AND
            (NOT bEjectBaseAlarm) AND (NOT bEjectModeAlarm) AND (NOT bCoreAlarm),
        bClampDone := bClampDone,
        bClampAlarm := bClampAlarm,
        bMoldOpened := bMoldOpened,
        bMoldClosed := bMoldClosed,
        bNozzleDone := bNozzleDone,
        bNozzleAlarm := bNozzleAlarm,
        bNozzleIned := bNozzleIned,
        bNozzleOuted := bNozzleOuted,
        bInjectDone := bInjectDone,
        bInjectAlarm := bInjectAlarm,
        bHeld := bHeld,
        bSuckBacked := bSuckBacked,
        bMeterDone := bMeterDone,
        bMeterAlarm := bMeterAlarm,
        bMetered := bMetered,
        bEjectDone := bEjectBaseDone,
        bEjectAlarm := bEjectBaseAlarm,
        bEjectIned := bEjectBaseIned,
        bEjectOuted := bEjectBaseOuted,
        bBusy => bAutoBusy,
        bDone => bAutoDone,
        bAlarm => bAutoAlarm,
        dwAlarmID => dwAutoAlarmID,
        uiActHint => uiAutoActHint,
        uiActTime => uiAutoActTime,
        uiCycleCount => uiAutoCycleCount,
        bClampStart => bAutoClampStart,
        bClampReset => bAutoClampReset,
        uiClampMode => uiAutoClampMode,
        bNozzleStart => bAutoNozzleStart,
        bNozzleReset => bAutoNozzleReset,
        uiNozzleMode => uiAutoNozzleMode,
        bInjectStart => bAutoInjectStart,
        bInjectReset => bAutoInjectReset,
        uiInjectMode => uiAutoInjectMode,
        bMeterStart => bAutoMeterStart,
        bMeterReset => bAutoMeterReset,
        bEjectStart => bAutoEjectStart,
        bEjectReset => bAutoEjectReset,
        uiEjectMode => uiAutoEjectMode
    );

    fbCommandComposer(
        stCommand := stCommand,                                             // 把最终机器命令送入命令合成层，统一收口公共复位与手动命令结构。
        stModeState := stModeState,                                         // 把本拍模式状态结构送入命令合成层，决定最终命令应由哪一类来源接管。
        bManualClampStart := bManualClampStart,                             // 把手动或调模路由结果中的合模启动命令送入命令合成层。
        uiManualClampMode := uiManualClampMode,                             // 把手动或调模路由结果中的合模模式号送入命令合成层。
        bManualMoldAdjustStart := bManualMoldAdjustStart,                   // 把手动或调模路由结果中的调模启动命令送入命令合成层。
        uiManualMoldAdjustMode := uiManualMoldAdjustMode,                   // 把手动或调模路由结果中的调模模式号送入命令合成层。
        bManualNozzleStart := bManualNozzleStart,                           // 把手动路由结果中的座台启动命令送入命令合成层。
        uiManualNozzleMode := uiManualNozzleMode,                           // 把手动路由结果中的座台模式号送入命令合成层。
        bManualInjectStart := bManualInjectStart,                           // 把手动路由结果中的射胶启动命令送入命令合成层。
        uiManualInjectMode := uiManualInjectMode,                           // 把手动路由结果中的射胶模式号送入命令合成层。
        bManualMeterStart := bManualMeterStart,                             // 把手动路由结果中的储料启动命令送入命令合成层。
        bManualEjectStart := bManualEjectStart,                             // 把手动路由结果中的基础托模启动命令送入命令合成层。
        uiManualEjectMode := uiManualEjectMode,                             // 把手动路由结果中的基础托模模式号送入命令合成层。
        bManualEjectModeStart := bManualEjectModeStart,                     // 把手动路由结果中的托模组合模式启动命令送入命令合成层。
        uiManualEjectPatternMode := uiManualEjectPatternMode,               // 把手动路由结果中的托模组合模式号送入命令合成层。
        uiManualEjectTimes := uiManualEjectTimes,                           // 把手动路由结果中的托模组合次数送入命令合成层。
        bManualCoreStart := bManualCoreStart,                               // 把手动路由结果中的中子启动命令送入命令合成层。
        uiManualCoreMode := uiManualCoreMode,                               // 把手动路由结果中的中子模式号送入命令合成层。
        bAutoClampStart := bAutoClampStart,                                 // 把自动流程输出中的合模启动命令送入命令合成层。
        bAutoClampReset := bAutoClampReset,                                 // 把自动流程输出中的合模复位命令送入命令合成层。
        uiAutoClampMode := uiAutoClampMode,                                 // 把自动流程输出中的合模模式号送入命令合成层。
        bAutoNozzleStart := bAutoNozzleStart,                               // 把自动流程输出中的座台启动命令送入命令合成层。
        bAutoNozzleReset := bAutoNozzleReset,                               // 把自动流程输出中的座台复位命令送入命令合成层。
        uiAutoNozzleMode := uiAutoNozzleMode,                               // 把自动流程输出中的座台模式号送入命令合成层。
        bAutoInjectStart := bAutoInjectStart,                               // 把自动流程输出中的射胶启动命令送入命令合成层。
        bAutoInjectReset := bAutoInjectReset,                               // 把自动流程输出中的射胶复位命令送入命令合成层。
        uiAutoInjectMode := uiAutoInjectMode,                               // 把自动流程输出中的射胶模式号送入命令合成层。
        bAutoMeterStart := bAutoMeterStart,                                 // 把自动流程输出中的储料启动命令送入命令合成层。
        bAutoMeterReset := bAutoMeterReset,                                 // 把自动流程输出中的储料复位命令送入命令合成层。
        bAutoEjectStart := bAutoEjectStart,                                 // 把自动流程输出中的基础托模启动命令送入命令合成层。
        bAutoEjectReset := bAutoEjectReset,                                 // 把自动流程输出中的基础托模复位命令送入命令合成层。
        uiAutoEjectMode := uiAutoEjectMode,                                 // 把自动流程输出中的基础托模模式号送入命令合成层。
        stModuleCommands => stModuleCommands,                               // 回收本拍合成出的最终模块命令集合，供执行模块统一消费。
        bUseEjectModeManual => bUseEjectModeManual                          // 回收当前托模是否切换到托模组合模式块的选择结果。
    );
END_IF;

(* 依次调用执行模块。 *)
fbClamp(
    ClampAxis := stClampAxis,
    bStart := stModuleCommands.bClampStart,
    bStop := stModeState.bGlobalStop,
    bEStop := stCommand.bEStop,
    bReset := stModuleCommands.bClampReset,
    bManualMode := stModeState.bManualModeActive,
    uiClampMode := stModuleCommands.uiClampMode,
    stClampPara := stPara.stClampPara,
    bOpenStop := stSensor.bOpenStop,
    bCloseLowPres := stSensor.bCloseLowPres,
    bCloseHighPres := stSensor.bCloseHighPres,
    bCloseStop := stSensor.bCloseStop,
    udiClampElecRulerVal := stSensor.udiClampElecRulerVal,
    uiClampPresElecRulerVal := stSensor.uiClampPresElecRulerVal,
    rClampActualPosition := stSensor.rClampActualPosition,
    rClampActualVelocity := stSensor.rClampActualVelocity,
    rClampActualPressure := stSensor.rClampActualPressure,
    bBusy => bClampBusy,
    bDone => bClampDone,
    bAlarm => bClampAlarm,
    dwAlarmID => dwClampAlarmID,
    uiActHint => uiClampActHint,
    uiActTime => uiClampActTime,
    bMoldOpened => bMoldOpened,
    bMoldClosed => bMoldClosed,
    aCoreAllow => aCoreAllowLocal
);

fbMoldAdjust(
    stMoldAdjustAxis := stMoldAdjustAxis,
    bStart := stModuleCommands.bMoldAdjustStart,
    bStop := stModeState.bGlobalStop OR (NOT (stModeState.bManualModeActive OR stModeState.bMoldAdjustModeActive)),
    bEStop := stCommand.bEStop,
    bReset := stModuleCommands.bMoldAdjustReset,
    (* 这里只在“机器手动模式”下把整个调模块切到手动点动。
       当机器处于“调模模式”时，仍允许 uiMoldAdjustMode=1/2 按工艺段自动进退，
       也允许 uiMoldAdjustMode=3/4 进入手动点动，因此这里不直接把调模模式映射为 bManualMode=TRUE。
    *)
    bManualMode := stModeState.bManualModeActive,
    uiMoldAdjustMode := stModuleCommands.uiMoldAdjustMode,
    stMoldAdjustPara := stPara.stMoldAdjustPara,
    bMoldAdjustInStop := stSensor.bMoldAdjustInStop,
    bMoldAdjustOutStop := stSensor.bMoldAdjustOutStop,
    uiClampPresElecRulerVal := stSensor.uiClampPresElecRulerVal,
    rMoldAdjustActualPosition := stSensor.rMoldAdjustActualPosition,
    rMoldAdjustActualVelocity := stSensor.rMoldAdjustActualVelocity,
    rMoldAdjustActualPressure := stSensor.rMoldAdjustActualPressure,
    bBusy => bMoldAdjustBusy,
    bDone => bMoldAdjustDone,
    bAlarm => bMoldAdjustAlarm,
    dwAlarmID => dwMoldAdjustAlarmID,
    uiActHint => uiMoldAdjustActHint,
    uiActTime => uiMoldAdjustActTime,
    bMoldAdjustIned => bMoldAdjustIned,
    bMoldAdjustOuted => bMoldAdjustOuted
);

fbNozzle(
    stNozzleAxis := stNozzleAxis,
    bStart := stModuleCommands.bNozzleStart,
    bStop := stModeState.bGlobalStop,
    bEStop := stCommand.bEStop,
    bReset := stModuleCommands.bNozzleReset,
    bManualMode := stModeState.bManualModeActive,
    uiNozzleMode := stModuleCommands.uiNozzleMode,
    stNozzlePara := stPara.stNozzlePara,
    bNozzleInStop := stSensor.bNozzleInStop,
    bNozzleOutStop := stSensor.bNozzleOutStop,
    udiNozzleElecRulerVal := stSensor.udiNozzleElecRulerVal,
    rNozzleActualPosition := stSensor.rNozzleActualPosition,
    rNozzleActualVelocity := stSensor.rNozzleActualVelocity,
    rNozzleActualPressure := stSensor.rNozzleActualPressure,
    bBusy => bNozzleBusy,
    bDone => bNozzleDone,
    bAlarm => bNozzleAlarm,
    dwAlarmID => dwNozzleAlarmID,
    uiActHint => uiNozzleActHint,
    uiActTime => uiNozzleActTime,
    bNozzleIned => bNozzleIned,
    bNozzleOuted => bNozzleOuted
);

fbInject(
    stInjectAxis := stInjectAxis,
    bStart := stModuleCommands.bInjectStart,
    bStop := stModeState.bGlobalStop,
    bEStop := stCommand.bEStop,
    bReset := stModuleCommands.bInjectReset,
    bManualMode := stModeState.bManualModeActive,
    uiInjectMode := stModuleCommands.uiInjectMode,
    stInjectPara := stPara.stInjectPara,
    bInjSeg1Stop := stSensor.bInjSeg1Stop,
    bInjSeg2Stop := stSensor.bInjSeg2Stop,
    bInjStop := stSensor.bInjStop,
    bSuckBackStop := stSensor.bSuckBackStop,
    udiInjElecRulerVal := stSensor.udiInjElecRulerVal,
    rInjectActualPosition := stSensor.rInjectActualPosition,
    rInjectActualVelocity := stSensor.rInjectActualVelocity,
    rInjectActualPressure := stSensor.rInjectActualPressure,
    bBusy => bInjectBusy,
    bDone => bInjectDone,
    bAlarm => bInjectAlarm,
    dwAlarmID => dwInjectAlarmID,
    uiActHint => uiInjectActHint,
    uiActTime => uiInjectActTime,
    bInjected => bInjected,
    bHeld => bHeld,
    bSuckBacked => bSuckBacked
);

fbMeter(
    stMeterAxis := stMeterAxis,
    bStart := stModuleCommands.bMeterStart,
    bStop := stModeState.bGlobalStop,
    bEStop := stCommand.bEStop,
    bReset := stModuleCommands.bMeterReset,
    bManualMode := stModeState.bManualModeActive,
    stMeterPara := stPara.stMeterPara,
    bMeterStop := stSensor.bMeterStop,
    udiInjElecRulerVal := stSensor.udiInjElecRulerVal,
    rMeterActualPosition := stSensor.rMeterActualPosition,
    rMeterActualVelocity := stSensor.rMeterActualVelocity,
    rMeterActualPressure := stSensor.rMeterActualPressure,
    bBusy => bMeterBusy,
    bDone => bMeterDone,
    bAlarm => bMeterAlarm,
    dwAlarmID => dwMeterAlarmID,
    uiActHint => uiMeterActHint,
    uiActTime => uiMeterActTime,
    bMetered => bMetered
);

fbEject(
    stEjectAxis := stEjectAxisBase,
    bStart := stModuleCommands.bEjectStart,
    bStop := stModeState.bGlobalStop OR bUseEjectModeManual,
    bEStop := stCommand.bEStop,
    bReset := stModuleCommands.bEjectReset,
    bManualMode := stModeState.bManualModeActive,
    uiEjectMode := stModuleCommands.uiEjectMode,
    stEjectPara := stPara.stEjectPara,
    bEjectInStop := stSensor.bEjectInStop,
    bEjectOutStop := stSensor.bEjectOutStop,
    udiEjectElecRulerVal := stSensor.udiEjectElecRulerVal,
    rEjectActualPosition := stSensor.rEjectActualPosition,
    rEjectActualVelocity := stSensor.rEjectActualVelocity,
    rEjectActualPressure := stSensor.rEjectActualPressure,
    bBusy => bEjectBaseBusy,
    bDone => bEjectBaseDone,
    bAlarm => bEjectBaseAlarm,
    dwAlarmID => dwEjectBaseAlarmID,
    uiActHint => uiEjectBaseActHint,
    uiActTime => uiEjectBaseActTime,
    bEjectIned => bEjectBaseIned,
    bEjectOuted => bEjectBaseOuted
);

fbEjectMode(
    stEjectAxis := stEjectAxisMode,
    bStart := stModuleCommands.bEjectModeStart,
    bStop := stModeState.bGlobalStop OR (NOT bUseEjectModeManual),
    bEStop := stCommand.bEStop,
    bReset := stModuleCommands.bEjectModeReset,
    uiEjectMode := stModuleCommands.uiEjectPatternMode,
    uiEjectTimes := stModuleCommands.uiEjectTimes,
    stEjectPara := stPara.stEjectPara,
    bEjectInStop := stSensor.bEjectInStop,
    bEjectOutStop := stSensor.bEjectOutStop,
    udiEjectElecRulerVal := stSensor.udiEjectElecRulerVal,
    rEjectActualPosition := stSensor.rEjectActualPosition,
    rEjectActualVelocity := stSensor.rEjectActualVelocity,
    rEjectActualPressure := stSensor.rEjectActualPressure,
    bBusy => bEjectModeBusy,
    bDone => bEjectModeDone,
    bAlarm => bEjectModeAlarm,
    dwAlarmID => dwEjectModeAlarmID,
    uiActHint => uiEjectModeActHint,
    uiActTime => uiEjectModeActTime,
    bEjectIned => bEjectModeIned,
    bEjectOuted => bEjectModeOuted
);

fbCore(
    stCoreAxis := stCoreAxis,
    bStart := stModuleCommands.bCoreStart,
    bStop := stModeState.bGlobalStop OR (NOT stModeState.bManualModeActive),
    bEStop := stCommand.bEStop,
    bReset := stModuleCommands.bCoreReset,
    bManualMode := stModeState.bManualModeActive,
    uiCoreMode := stModuleCommands.uiCoreMode,
    stCorePara := stPara.stCorePara,
    bCoreInStop := stSensor.bCoreInStop,
    bCoreOutStop := stSensor.bCoreOutStop,
    rCoreActualPosition := stSensor.rCoreActualPosition,
    rCoreActualVelocity := stSensor.rCoreActualVelocity,
    rCoreActualPressure := stSensor.rCoreActualPressure,
    bBusy => bCoreBusy,
    bDone => bCoreDone,
    bAlarm => bCoreAlarm,
    dwAlarmID => dwCoreAlarmID,
    uiActHint => uiCoreActHint,
    uiActTime => uiCoreActTime,
    bCoreIned => bCoreIned,
    bCoreOuted => bCoreOuted
);

(* 由主控层统一选择当前托模输出来源。 *)
IF bUseEjectModeManual THEN
    stEjectAxis := stEjectAxisMode;                       // 手动组合托模生效时，对外输出切换为 `FB_EjectMode` 的轴结果。
    bSelectedEjectBusy := bEjectModeBusy;                 // 手动组合托模生效时，托模 Busy 状态取自 `FB_EjectMode`。
    bSelectedEjectDone := bEjectModeDone;                 // 手动组合托模生效时，托模 Done 状态取自 `FB_EjectMode`。
    bSelectedEjectAlarm := bEjectModeAlarm;               // 手动组合托模生效时，托模 Alarm 状态取自 `FB_EjectMode`。
    dwSelectedEjectAlarmID := dwEjectModeAlarmID;         // 手动组合托模生效时，托模报警码取自 `FB_EjectMode`。
    uiSelectedEjectActHint := uiEjectModeActHint;         // 手动组合托模生效时，托模动作提示号取自 `FB_EjectMode`。
    uiSelectedEjectActTime := uiEjectModeActTime;         // 手动组合托模生效时，托模动作时间取自 `FB_EjectMode`。
    bSelectedEjectIned := bEjectModeIned;                 // 手动组合托模生效时，托模内位到位状态取自 `FB_EjectMode`。
    bSelectedEjectOuted := bEjectModeOuted;               // 手动组合托模生效时，托模外位到位状态取自 `FB_EjectMode`。
ELSE
    stEjectAxis := stEjectAxisBase;                       // 未启用手动组合托模时，对外输出保持为基础托模块的轴结果。
    bSelectedEjectBusy := bEjectBaseBusy;                 // 未启用手动组合托模时，托模 Busy 状态取自基础托模块。
    bSelectedEjectDone := bEjectBaseDone;                 // 未启用手动组合托模时，托模 Done 状态取自基础托模块。
    bSelectedEjectAlarm := bEjectBaseAlarm;               // 未启用手动组合托模时，托模 Alarm 状态取自基础托模块。
    dwSelectedEjectAlarmID := dwEjectBaseAlarmID;         // 未启用手动组合托模时，托模报警码取自基础托模块。
    uiSelectedEjectActHint := uiEjectBaseActHint;         // 未启用手动组合托模时，托模动作提示号取自基础托模块。
    uiSelectedEjectActTime := uiEjectBaseActTime;         // 未启用手动组合托模时，托模动作时间取自基础托模块。
    bSelectedEjectIned := bEjectBaseIned;                 // 未启用手动组合托模时，托模内位到位状态取自基础托模块。
    bSelectedEjectOuted := bEjectBaseOuted;               // 未启用手动组合托模时，托模外位到位状态取自基础托模块。
END_IF;

FOR uiIndex := 1 TO 8 DO
    aCoreAllow[uiIndex] := aCoreAllowLocal[uiIndex];      // 逐路把合模块给出的中子允许位复制到对外输出数组。
END_FOR;

(* 机器级状态汇总。 *)
fbStatusAggregator(
    stCommand := stCommand,                           // 把最终机器命令送入状态汇总层，回写当前机器模式号。
    stSensor := stSensor,                             // 把现场传感器边界送入状态汇总层，计算自动准备就绪综合结果。
    stModeState := stModeState,                       // 把本拍模式状态结构送入状态汇总层，回写当前模式与自动模式号。
    bAutoBusy := bAutoBusy,                           // 把自动流程 Busy 状态送入状态汇总层。
    bAutoDone := bAutoDone,                           // 把自动流程 Done 状态送入状态汇总层。
    bAutoAlarm := bAutoAlarm,                         // 把自动流程 Alarm 状态送入状态汇总层。
    dwAutoAlarmID := dwAutoAlarmID,                   // 把自动流程报警码送入状态汇总层。
    uiAutoActHint := uiAutoActHint,                   // 把自动流程动作提示号送入状态汇总层。
    uiAutoActTime := uiAutoActTime,                   // 把自动流程动作持续时间送入状态汇总层。
    uiAutoCycleCount := uiAutoCycleCount,             // 把自动流程累计循环次数送入状态汇总层。
    bClampBusy := bClampBusy,                         // 把合模块 Busy 状态送入状态汇总层。
    bClampDone := bClampDone,                         // 把合模块 Done 状态送入状态汇总层。
    bClampAlarm := bClampAlarm,                       // 把合模块 Alarm 状态送入状态汇总层。
    dwClampAlarmID := dwClampAlarmID,                 // 把合模块报警码送入状态汇总层。
    uiClampActHint := uiClampActHint,                 // 把合模块动作提示号送入状态汇总层。
    uiClampActTime := uiClampActTime,                 // 把合模块动作持续时间送入状态汇总层。
    bMoldOpened := bMoldOpened,                       // 把开模到位状态送入状态汇总层。
    bMoldClosed := bMoldClosed,                       // 把合模到位状态送入状态汇总层。
    bMoldAdjustBusy := bMoldAdjustBusy,               // 把调模块 Busy 状态送入状态汇总层。
    bMoldAdjustDone := bMoldAdjustDone,               // 把调模块 Done 状态送入状态汇总层。
    bMoldAdjustAlarm := bMoldAdjustAlarm,             // 把调模块 Alarm 状态送入状态汇总层。
    dwMoldAdjustAlarmID := dwMoldAdjustAlarmID,       // 把调模块报警码送入状态汇总层。
    uiMoldAdjustActHint := uiMoldAdjustActHint,       // 把调模块动作提示号送入状态汇总层。
    uiMoldAdjustActTime := uiMoldAdjustActTime,       // 把调模块动作持续时间送入状态汇总层。
    bMoldAdjustIned := bMoldAdjustIned,               // 把调模进到位状态送入状态汇总层。
    bMoldAdjustOuted := bMoldAdjustOuted,             // 把调模退到位状态送入状态汇总层。
    bNozzleBusy := bNozzleBusy,                       // 把座台模块 Busy 状态送入状态汇总层。
    bNozzleDone := bNozzleDone,                       // 把座台模块 Done 状态送入状态汇总层。
    bNozzleAlarm := bNozzleAlarm,                     // 把座台模块 Alarm 状态送入状态汇总层。
    dwNozzleAlarmID := dwNozzleAlarmID,               // 把座台模块报警码送入状态汇总层。
    uiNozzleActHint := uiNozzleActHint,               // 把座台模块动作提示号送入状态汇总层。
    uiNozzleActTime := uiNozzleActTime,               // 把座台模块动作持续时间送入状态汇总层。
    bNozzleIned := bNozzleIned,                       // 把座进到位状态送入状态汇总层。
    bNozzleOuted := bNozzleOuted,                     // 把座退到位状态送入状态汇总层。
    bInjectBusy := bInjectBusy,                       // 把射胶模块 Busy 状态送入状态汇总层。
    bInjectDone := bInjectDone,                       // 把射胶模块 Done 状态送入状态汇总层。
    bInjectAlarm := bInjectAlarm,                     // 把射胶模块 Alarm 状态送入状态汇总层。
    dwInjectAlarmID := dwInjectAlarmID,               // 把射胶模块报警码送入状态汇总层。
    uiInjectActHint := uiInjectActHint,               // 把射胶模块动作提示号送入状态汇总层。
    uiInjectActTime := uiInjectActTime,               // 把射胶模块动作持续时间送入状态汇总层。
    bInjected := bInjected,                           // 把射出完成状态送入状态汇总层。
    bHeld := bHeld,                                   // 把保压完成状态送入状态汇总层。
    bSuckBacked := bSuckBacked,                       // 把射退完成状态送入状态汇总层。
    bMeterBusy := bMeterBusy,                         // 把储料模块 Busy 状态送入状态汇总层。
    bMeterDone := bMeterDone,                         // 把储料模块 Done 状态送入状态汇总层。
    bMeterAlarm := bMeterAlarm,                       // 把储料模块 Alarm 状态送入状态汇总层。
    dwMeterAlarmID := dwMeterAlarmID,                 // 把储料模块报警码送入状态汇总层。
    uiMeterActHint := uiMeterActHint,                 // 把储料模块动作提示号送入状态汇总层。
    uiMeterActTime := uiMeterActTime,                 // 把储料模块动作持续时间送入状态汇总层。
    bMetered := bMetered,                             // 把储料完成状态送入状态汇总层。
    bUseEjectModeManual := bUseEjectModeManual,       // 把当前托模来源选择结果送入状态汇总层。
    bSelectedEjectBusy := bSelectedEjectBusy,         // 把当前托模来源 Busy 状态送入状态汇总层。
    bSelectedEjectDone := bSelectedEjectDone,         // 把当前托模来源 Done 状态送入状态汇总层。
    bSelectedEjectAlarm := bSelectedEjectAlarm,       // 把当前托模来源 Alarm 状态送入状态汇总层。
    dwSelectedEjectAlarmID := dwSelectedEjectAlarmID, // 把当前托模来源报警码送入状态汇总层。
    uiSelectedEjectActHint := uiSelectedEjectActHint, // 把当前托模来源动作提示号送入状态汇总层。
    uiSelectedEjectActTime := uiSelectedEjectActTime, // 把当前托模来源动作持续时间送入状态汇总层。
    bSelectedEjectIned := bSelectedEjectIned,         // 把当前托模来源内位到位状态送入状态汇总层。
    bSelectedEjectOuted := bSelectedEjectOuted,       // 把当前托模来源外位到位状态送入状态汇总层。
    bCoreBusy := bCoreBusy,                           // 把中子模块 Busy 状态送入状态汇总层。
    bCoreDone := bCoreDone,                           // 把中子模块 Done 状态送入状态汇总层。
    bCoreAlarm := bCoreAlarm,                         // 把中子模块 Alarm 状态送入状态汇总层。
    dwCoreAlarmID := dwCoreAlarmID,                   // 把中子模块报警码送入状态汇总层。
    uiCoreActHint := uiCoreActHint,                   // 把中子模块动作提示号送入状态汇总层。
    uiCoreActTime := uiCoreActTime,                   // 把中子模块动作持续时间送入状态汇总层。
    bCoreIned := bCoreIned,                           // 把中子进到位状态送入状态汇总层。
    bCoreOuted := bCoreOuted,                         // 把中子退到位状态送入状态汇总层。
    stStatus => stStatus                              // 回收汇总后的机器级总状态，供顶层与 HMI 统一读取。
);
END_FUNCTION_BLOCK

(* ---- FB_MachineModeResolver.st ---- *)
(*
  FB_MachineModeResolver 功能块
  功能：
  1. 统一解析当前机器模式，并生成主控内部使用的模式状态结构。
  2. 把切模检测、自动模式号换算和全局停止位都收口到同一层。
  3. 当前块只做模式解析，不处理任何模块命令与状态汇总。
*)
FUNCTION_BLOCK FB_MachineModeResolver
VAR_INPUT
    stCommand: ST_MachineCommand;        // 顶层下发的最终机器命令；当前块只消费其中公共模式与停机命令。
END_VAR
VAR_OUTPUT
    stModeState: ST_MachineModeState;    // 当前扫描周期解析出的模式状态结构；供主控后续命令合成与状态汇总使用。
END_VAR
VAR
    uiLastMachineMode: UINT := 0;        // 上一扫描周期保存的机器模式号；用于与当前模式比较判断是否切模。
END_VAR

stModeState.bManualModeActive := (stCommand.uiMachineMode = 1);                                     // 模式号为 1 时，主控标记当前进入手动模式。
stModeState.bMoldAdjustModeActive := (stCommand.uiMachineMode = 4);                                 // 模式号为 4 时，主控标记当前进入调模模式。
stModeState.bSemiAutoModeActive := (stCommand.uiMachineMode = 2);                                   // 模式号为 2 时，主控标记当前进入半自动模式。
stModeState.bFullAutoModeActive := (stCommand.uiMachineMode = 3);                                   // 模式号为 3 时，主控标记当前进入全自动模式。
stModeState.bModeChanged := (uiLastMachineMode <> stCommand.uiMachineMode);                         // 当前模式号与上一拍不同则认为发生了模式切换。
uiLastMachineMode := stCommand.uiMachineMode;                                                        // 保存本拍模式号，供下一拍继续检测是否切模。
stModeState.bGlobalStop := stCommand.bStop OR (stCommand.uiMachineMode = 0) OR stModeState.bModeChanged; // 停止命令、停机模式或切模保护任一出现，都统一触发主控总停止。

IF stModeState.bSemiAutoModeActive THEN                                                              // 半自动模式时，把自动流程工作模式解析为 1。
    stModeState.uiResolvedAutoMode := 1;                                                             // `FB_AutoCycle` 用 1 表示半自动。
ELSIF stModeState.bFullAutoModeActive THEN                                                           // 全自动模式时，把自动流程工作模式解析为 2。
    stModeState.uiResolvedAutoMode := 2;                                                             // `FB_AutoCycle` 用 2 表示全自动。
ELSE
    stModeState.uiResolvedAutoMode := 0;                                                             // 非自动模式时，明确告知自动流程当前不参与调度。
END_IF;
END_FUNCTION_BLOCK

(* ---- FB_MachineStatusAggregator.st ---- *)
(*
  FB_MachineStatusAggregator 功能块
  功能：
  1. 把自动流程、各执行模块和模式解析结果汇总为统一的机器级状态输出。
  2. 统一决定整机 Busy/Done/Alarm、当前动作提示与最高优先级报警号。
  3. 当前块只负责状态汇总，不直接驱动任何执行模块。
*)
FUNCTION_BLOCK FB_MachineStatusAggregator
VAR_INPUT
    stCommand: ST_MachineCommand;            // 顶层下发的最终机器命令；当前块只消费其中当前机器模式号。
    stSensor: ST_MachineSensor;              // 顶层采集的现场条件与传感器；当前块用于计算自动准备就绪状态。
    stModeState: ST_MachineModeState;        // 当前扫描周期解析出的模式状态结构；当前块用于汇总当前模式与自动模式号。

    (* 自动流程状态。 *)
    bAutoBusy: BOOL;                         // 自动流程 Busy 状态。
    bAutoDone: BOOL;                         // 自动流程 Done 状态。
    bAutoAlarm: BOOL;                        // 自动流程 Alarm 状态。
    dwAutoAlarmID: DWORD;                    // 自动流程报警码。
    uiAutoActHint: UINT;                     // 自动流程动作提示号。
    uiAutoActTime: UINT;                     // 自动流程动作持续时间。
    uiAutoCycleCount: UINT;                  // 自动流程累计循环次数。

    (* 合模块状态。 *)
    bClampBusy: BOOL;                        // 合模块 Busy 状态。
    bClampDone: BOOL;                        // 合模块 Done 状态。
    bClampAlarm: BOOL;                       // 合模块 Alarm 状态。
    dwClampAlarmID: DWORD;                   // 合模块报警码。
    uiClampActHint: UINT;                    // 合模块动作提示号。
    uiClampActTime: UINT;                    // 合模块动作持续时间。
    bMoldOpened: BOOL;                       // 合模块开模到位状态。
    bMoldClosed: BOOL;                       // 合模块合模到位状态。

    (* 调模块状态。 *)
    bMoldAdjustBusy: BOOL;                   // 调模块 Busy 状态。
    bMoldAdjustDone: BOOL;                   // 调模块 Done 状态。
    bMoldAdjustAlarm: BOOL;                  // 调模块 Alarm 状态。
    dwMoldAdjustAlarmID: DWORD;              // 调模块报警码。
    uiMoldAdjustActHint: UINT;               // 调模块动作提示号。
    uiMoldAdjustActTime: UINT;               // 调模块动作持续时间。
    bMoldAdjustIned: BOOL;                   // 调模块进到位状态。
    bMoldAdjustOuted: BOOL;                  // 调模块退到位状态。

    (* 座台模块状态。 *)
    bNozzleBusy: BOOL;                       // 座台模块 Busy 状态。
    bNozzleDone: BOOL;                       // 座台模块 Done 状态。
    bNozzleAlarm: BOOL;                      // 座台模块 Alarm 状态。
    dwNozzleAlarmID: DWORD;                  // 座台模块报警码。
    uiNozzleActHint: UINT;                   // 座台模块动作提示号。
    uiNozzleActTime: UINT;                   // 座台模块动作持续时间。
    bNozzleIned: BOOL;                       // 座台模块进到位状态。
    bNozzleOuted: BOOL;                      // 座台模块退到位状态。

    (* 射胶模块状态。 *)
    bInjectBusy: BOOL;                       // 射胶模块 Busy 状态。
    bInjectDone: BOOL;                       // 射胶模块 Done 状态。
    bInjectAlarm: BOOL;                      // 射胶模块 Alarm 状态。
    dwInjectAlarmID: DWORD;                  // 射胶模块报警码。
    uiInjectActHint: UINT;                   // 射胶模块动作提示号。
    uiInjectActTime: UINT;                   // 射胶模块动作持续时间。
    bInjected: BOOL;                         // 射胶模块射出完成状态。
    bHeld: BOOL;                             // 射胶模块保压完成状态。
    bSuckBacked: BOOL;                       // 射胶模块射退完成状态。

    (* 储料模块状态。 *)
    bMeterBusy: BOOL;                        // 储料模块 Busy 状态。
    bMeterDone: BOOL;                        // 储料模块 Done 状态。
    bMeterAlarm: BOOL;                       // 储料模块 Alarm 状态。
    dwMeterAlarmID: DWORD;                   // 储料模块报警码。
    uiMeterActHint: UINT;                    // 储料模块动作提示号。
    uiMeterActTime: UINT;                    // 储料模块动作持续时间。
    bMetered: BOOL;                          // 储料模块储料完成状态。

    (* 当前被选中的托模来源状态。 *)
    bUseEjectModeManual: BOOL;               // TRUE=当前托模输出来自托模组合模式块，而不是基础托模块。
    bSelectedEjectBusy: BOOL;                // 当前被选中的托模来源 Busy 状态。
    bSelectedEjectDone: BOOL;                // 当前被选中的托模来源 Done 状态。
    bSelectedEjectAlarm: BOOL;               // 当前被选中的托模来源 Alarm 状态。
    dwSelectedEjectAlarmID: DWORD;           // 当前被选中的托模来源报警码。
    uiSelectedEjectActHint: UINT;            // 当前被选中的托模来源动作提示号。
    uiSelectedEjectActTime: UINT;            // 当前被选中的托模来源动作持续时间。
    bSelectedEjectIned: BOOL;                // 当前被选中的托模来源内位到位状态。
    bSelectedEjectOuted: BOOL;               // 当前被选中的托模来源外位到位状态。

    (* 中子模块状态。 *)
    bCoreBusy: BOOL;                         // 中子模块 Busy 状态。
    bCoreDone: BOOL;                         // 中子模块 Done 状态。
    bCoreAlarm: BOOL;                        // 中子模块 Alarm 状态。
    dwCoreAlarmID: DWORD;                    // 中子模块报警码。
    uiCoreActHint: UINT;                     // 中子模块动作提示号。
    uiCoreActTime: UINT;                     // 中子模块动作持续时间。
    bCoreIned: BOOL;                         // 中子模块进到位状态。
    bCoreOuted: BOOL;                        // 中子模块退到位状态。
END_VAR
VAR_OUTPUT
    stStatus: ST_MachineStatus;             // 汇总后的机器级总状态；供 HMI、上位机和顶层逻辑统一读取。
END_VAR
VAR
    bAutoReadyLocal: BOOL := FALSE;         // 自动循环可启动条件综合结果；最终写入 `stStatus.bAutoReady`。
END_VAR

bAutoReadyLocal := stSensor.bDoorClosed AND stSensor.bHydReady AND                           // 自动准备就绪必须满足门已关和液压已就绪两项基础前提。
    stSensor.bSystemNoAlarm AND (NOT bClampAlarm) AND (NOT bMoldAdjustAlarm) AND            // 自动准备就绪还要求系统级与合模/调模块无报警。
    (NOT bNozzleAlarm) AND (NOT bInjectAlarm) AND (NOT bMeterAlarm) AND                      // 自动准备就绪还要求座台/射胶/储料模块无报警。
    (NOT bSelectedEjectAlarm) AND (NOT bCoreAlarm) AND (NOT bAutoAlarm);                     // 自动准备就绪还要求托模/中子/自动流程本身均无报警。

stStatus.uiMachineMode := stCommand.uiMachineMode;                               // 回写当前机器模式号，供 HMI 与上位机直接读取。
stStatus.bManualModeActive := stModeState.bManualModeActive;                     // 回写当前是否处于手动模式。
stStatus.bMoldAdjustModeActive := stModeState.bMoldAdjustModeActive;             // 回写当前是否处于调模模式。
stStatus.bSemiAutoModeActive := stModeState.bSemiAutoModeActive;                 // 回写当前是否处于半自动模式。
stStatus.bFullAutoModeActive := stModeState.bFullAutoModeActive;                 // 回写当前是否处于全自动模式。
stStatus.bAutoReady := bAutoReadyLocal;                                          // 回写自动准备就绪综合结果。
stStatus.uiCycleCount := uiAutoCycleCount;                                       // 回写自动循环累计次数。

stStatus.bAutoBusy := bAutoBusy;                                                 // 回写自动流程 Busy 状态。
stStatus.bAutoDone := bAutoDone;                                                 // 回写自动流程 Done 状态。
stStatus.bAutoAlarm := bAutoAlarm;                                               // 回写自动流程 Alarm 状态。
stStatus.dwAutoAlarmID := dwAutoAlarmID;                                         // 回写自动流程报警码。

stStatus.bClampBusy := bClampBusy;                                               // 回写合模块 Busy 状态。
stStatus.bClampDone := bClampDone;                                               // 回写合模块 Done 状态。
stStatus.bClampAlarm := bClampAlarm;                                             // 回写合模块 Alarm 状态。
stStatus.dwClampAlarmID := dwClampAlarmID;                                       // 回写合模块报警码。
stStatus.bMoldOpened := bMoldOpened;                                             // 回写开模到位状态。
stStatus.bMoldClosed := bMoldClosed;                                             // 回写合模到位状态。

stStatus.bMoldAdjustBusy := bMoldAdjustBusy;                                     // 回写调模块 Busy 状态。
stStatus.bMoldAdjustDone := bMoldAdjustDone;                                     // 回写调模块 Done 状态。
stStatus.bMoldAdjustAlarm := bMoldAdjustAlarm;                                   // 回写调模块 Alarm 状态。
stStatus.dwMoldAdjustAlarmID := dwMoldAdjustAlarmID;                             // 回写调模块报警码。
stStatus.bMoldAdjustIned := bMoldAdjustIned;                                     // 回写调模进到位状态。
stStatus.bMoldAdjustOuted := bMoldAdjustOuted;                                   // 回写调模退到位状态。

stStatus.bNozzleBusy := bNozzleBusy;                                             // 回写座台模块 Busy 状态。
stStatus.bNozzleDone := bNozzleDone;                                             // 回写座台模块 Done 状态。
stStatus.bNozzleAlarm := bNozzleAlarm;                                           // 回写座台模块 Alarm 状态。
stStatus.dwNozzleAlarmID := dwNozzleAlarmID;                                     // 回写座台模块报警码。
stStatus.bNozzleIned := bNozzleIned;                                             // 回写座进到位状态。
stStatus.bNozzleOuted := bNozzleOuted;                                           // 回写座退到位状态。

stStatus.bInjectBusy := bInjectBusy;                                             // 回写射胶模块 Busy 状态。
stStatus.bInjectDone := bInjectDone;                                             // 回写射胶模块 Done 状态。
stStatus.bInjectAlarm := bInjectAlarm;                                           // 回写射胶模块 Alarm 状态。
stStatus.dwInjectAlarmID := dwInjectAlarmID;                                     // 回写射胶模块报警码。
stStatus.bInjected := bInjected;                                                 // 回写射出完成状态。
stStatus.bHeld := bHeld;                                                         // 回写保压完成状态。
stStatus.bSuckBacked := bSuckBacked;                                             // 回写射退完成状态。

stStatus.bMeterBusy := bMeterBusy;                                               // 回写储料模块 Busy 状态。
stStatus.bMeterDone := bMeterDone;                                               // 回写储料模块 Done 状态。
stStatus.bMeterAlarm := bMeterAlarm;                                             // 回写储料模块 Alarm 状态。
stStatus.dwMeterAlarmID := dwMeterAlarmID;                                       // 回写储料模块报警码。
stStatus.bMetered := bMetered;                                                   // 回写储料完成状态。

stStatus.bEjectModeSelected := bUseEjectModeManual;                              // 回写当前托模输出是否来自托模组合模式块。
stStatus.bEjectBusy := bSelectedEjectBusy;                                       // 回写当前托模来源 Busy 状态。
stStatus.bEjectDone := bSelectedEjectDone;                                       // 回写当前托模来源 Done 状态。
stStatus.bEjectAlarm := bSelectedEjectAlarm;                                     // 回写当前托模来源 Alarm 状态。
stStatus.dwEjectAlarmID := dwSelectedEjectAlarmID;                               // 回写当前托模来源报警码。
stStatus.bEjectIned := bSelectedEjectIned;                                       // 回写当前托模来源内位到位状态。
stStatus.bEjectOuted := bSelectedEjectOuted;                                     // 回写当前托模来源外位到位状态。

stStatus.bCoreBusy := bCoreBusy;                                                 // 回写中子模块 Busy 状态。
stStatus.bCoreDone := bCoreDone;                                                 // 回写中子模块 Done 状态。
stStatus.bCoreAlarm := bCoreAlarm;                                               // 回写中子模块 Alarm 状态。
stStatus.dwCoreAlarmID := dwCoreAlarmID;                                         // 回写中子模块报警码。
stStatus.bCoreIned := bCoreIned;                                                 // 回写中子进到位状态。
stStatus.bCoreOuted := bCoreOuted;                                               // 回写中子退到位状态。

stStatus.bMachineBusy := bAutoBusy OR bClampBusy OR bMoldAdjustBusy OR bNozzleBusy OR bInjectBusy OR // 汇总整机 Busy 状态。
    bMeterBusy OR bSelectedEjectBusy OR bCoreBusy;

IF stModeState.uiResolvedAutoMode > 0 THEN
    stStatus.bMachineDone := bAutoDone;                                           // 自动模式下，整机 Done 直接跟随自动流程 Done。
ELSE
    stStatus.bMachineDone := bClampDone OR bMoldAdjustDone OR bNozzleDone OR bInjectDone OR // 非自动模式下，只要任一模块完成就对外回写 Done。
        bMeterDone OR bSelectedEjectDone OR bCoreDone;
END_IF;

stStatus.bMachineAlarm := bAutoAlarm OR bClampAlarm OR bMoldAdjustAlarm OR bNozzleAlarm OR // 汇总整机 Alarm 状态。
    bInjectAlarm OR bMeterAlarm OR bSelectedEjectAlarm OR bCoreAlarm;

IF bAutoAlarm THEN
    stStatus.dwMachineAlarmID := dwAutoAlarmID;                                   // 自动流程报警优先作为整机最高优先级报警号。
ELSIF bClampAlarm THEN
    stStatus.dwMachineAlarmID := dwClampAlarmID;                                  // 合模块报警次优先作为整机报警号。
ELSIF bMoldAdjustAlarm THEN
    stStatus.dwMachineAlarmID := dwMoldAdjustAlarmID;                             // 调模块报警作为整机报警号。
ELSIF bNozzleAlarm THEN
    stStatus.dwMachineAlarmID := dwNozzleAlarmID;                                 // 座台模块报警作为整机报警号。
ELSIF bInjectAlarm THEN
    stStatus.dwMachineAlarmID := dwInjectAlarmID;                                 // 射胶模块报警作为整机报警号。
ELSIF bMeterAlarm THEN
    stStatus.dwMachineAlarmID := dwMeterAlarmID;                                  // 储料模块报警作为整机报警号。
ELSIF bSelectedEjectAlarm THEN
    stStatus.dwMachineAlarmID := dwSelectedEjectAlarmID;                          // 当前托模来源报警作为整机报警号。
ELSIF bCoreAlarm THEN
    stStatus.dwMachineAlarmID := dwCoreAlarmID;                                   // 中子模块报警作为整机报警号。
ELSE
    stStatus.dwMachineAlarmID := DWORD#0;                                         // 无报警时清空整机报警号。
END_IF;

(* 当前动作提示优先显示自动流程；若不在自动流程中，则显示当前实际运行的模块。 *)
stStatus.uiMachineActHint := 0;                                                   // 每拍先清空整机动作提示号，随后按优先级回填。
stStatus.uiMachineActTime := 0;                                                   // 每拍先清空整机动作持续时间，随后按优先级回填。

IF (stModeState.uiResolvedAutoMode > 0) AND (bAutoBusy OR bAutoDone OR bAutoAlarm) THEN
    stStatus.uiMachineActHint := uiAutoActHint;                                   // 自动模式有效且自动流程正在运行时，优先显示自动流程动作提示。
    stStatus.uiMachineActTime := uiAutoActTime;                                   // 自动模式有效且自动流程正在运行时，优先显示自动流程动作时间。
ELSIF bClampBusy OR bClampDone OR bClampAlarm THEN
    stStatus.uiMachineActHint := uiClampActHint;                                  // 否则优先显示合模块动作提示。
    stStatus.uiMachineActTime := uiClampActTime;                                  // 否则优先显示合模块动作时间。
ELSIF bMoldAdjustBusy OR bMoldAdjustDone OR bMoldAdjustAlarm THEN
    stStatus.uiMachineActHint := uiMoldAdjustActHint;                             // 再否则显示调模块动作提示。
    stStatus.uiMachineActTime := uiMoldAdjustActTime;                             // 再否则显示调模块动作时间。
ELSIF bNozzleBusy OR bNozzleDone OR bNozzleAlarm THEN
    stStatus.uiMachineActHint := uiNozzleActHint;                                 // 再否则显示座台模块动作提示。
    stStatus.uiMachineActTime := uiNozzleActTime;                                 // 再否则显示座台模块动作时间。
ELSIF bInjectBusy OR bInjectDone OR bInjectAlarm THEN
    stStatus.uiMachineActHint := uiInjectActHint;                                 // 再否则显示射胶模块动作提示。
    stStatus.uiMachineActTime := uiInjectActTime;                                 // 再否则显示射胶模块动作时间。
ELSIF bMeterBusy OR bMeterDone OR bMeterAlarm THEN
    stStatus.uiMachineActHint := uiMeterActHint;                                  // 再否则显示储料模块动作提示。
    stStatus.uiMachineActTime := uiMeterActTime;                                  // 再否则显示储料模块动作时间。
ELSIF bSelectedEjectBusy OR bSelectedEjectDone OR bSelectedEjectAlarm THEN
    stStatus.uiMachineActHint := uiSelectedEjectActHint;                          // 再否则显示当前托模来源动作提示。
    stStatus.uiMachineActTime := uiSelectedEjectActTime;                          // 再否则显示当前托模来源动作时间。
ELSIF bCoreBusy OR bCoreDone OR bCoreAlarm THEN
    stStatus.uiMachineActHint := uiCoreActHint;                                   // 最后显示中子模块动作提示。
    stStatus.uiMachineActTime := uiCoreActTime;                                   // 最后显示中子模块动作时间。
END_IF;
END_FUNCTION_BLOCK

(* ---- PRG_MachineController.st ---- *)
(*
  PRG_MachineController 程序
  状态：兼容占位，禁止继续绑定到 PLC 任务。

  原因：
  1. 机器主控已经统一收口到 `PRG_MainControl`。
  2. 若本程序与 `PRG_MainControl` 同时执行，会导致 `gvl_fbMachineController`
     在同一扫描周期被重复调用，破坏状态机时序。
*)
PROGRAM PRG_MachineController
VAR
END_VAR

(* 兼容占位：无执行逻辑。请在工程任务配置中只保留 `PRG_MainControl`。 *)
END_PROGRAM

(* ---- PRG_MainControl.st ---- *)
(*
  PRG_MainControl 程序
  功能：
  1. 作为 PLC 工程唯一有效的主任务入口，统一调度 HMI 参数同步、面板调度、命令仲裁、顶层温控和机器主控。
  2. 本程序必须绑定到 1ms 基础任务；工艺逻辑由本程序在顶层生成固定 10ms 节拍后送给 `FB_MachineController`。
  3. 温控块 `FB_EK312` 必须由本程序在顶层直接调用，并由本程序在顶层生成固定 100ms 节拍后送给温控块刷新计算。
  4. 所有共享数据都通过 `全局变量\GlobalVars.st` 访问，不再拆分到多个顶层入口。

  维护要求：
  1. 工程任务配置只应绑定本程序，且基础周期固定为 1ms。
  2. 任何涉及主控流程、接口或架构的改动，都必须同步更新 3 份 MD 文档。
*)
PROGRAM PRG_MainControl
VAR
    (* `PRG_MainControl` 必须绑定到 1ms 基础任务；
       工艺逻辑按 10 拍执行一次，形成固定 10ms 逻辑节拍；
       温控系统按 100 拍执行一次，形成固定 100ms 逻辑节拍。
    *)
    uiLogicTickDiv: UINT := 0;                    // 10ms 逻辑节拍分频计数器，按 1ms 基础调用累加到第 10 拍后清零。
    bLogicTick10ms: BOOL := FALSE;                // TRUE=当前扫描周期命中一次 10ms 逻辑拍，允许主控刷新模式路由和自动流程。
    uiTempTickDiv: UINT := 0;                     // 100ms 温控节拍分频计数器，按 1ms 逻辑拍累加到第 100 拍后清零。
    bTempTick100ms: BOOL := FALSE;               // TRUE=当前扫描周期命中一次 100ms 逻辑拍，允许温控系统刷新一轮计算。
    stBaseCommandSnapshot: ST_MachineCommand;     // 当前扫描周期仲裁前的基础机器命令快照；用于保留外部入口写入的公共启动/停止/复位命令。
END_VAR

(* 基础调用周期固定按 1ms 设计；
   这里在顶层统一生成 10ms 工艺节拍和 100ms 温控节拍，
   让执行模块与其内部轴层仍然保持每拍 1ms 调用。
*)
bLogicTick10ms := FALSE;                        // 先把 10ms 节拍标志清零，只有命中分频点时才在当前扫描周期拉高一次。
IF uiLogicTickDiv >= 9 THEN                     // 当 1ms 基础拍累计满 10 次时，输出一次 10ms 逻辑节拍。
    uiLogicTickDiv := 0;                        // 10ms 分频计数器清零，开始统计下一轮 10ms 周期。
    bLogicTick10ms := TRUE;                     // 标记本扫描周期允许刷新一次主控工艺逻辑。
ELSE
    uiLogicTickDiv := uiLogicTickDiv + 1;       // 尚未达到 10ms 时继续累加 1ms 基础拍计数。
END_IF;

bTempTick100ms := FALSE;                        // 先把 100ms 节拍标志清零，只有命中分频点时才在当前扫描周期拉高一次。
IF uiTempTickDiv >= 99 THEN                     // 当 1ms 基础拍累计满 100 次时，输出一次 100ms 逻辑节拍。
    uiTempTickDiv := 0;                         // 100ms 分频计数器清零，开始统计下一轮 100ms 周期。
    bTempTick100ms := TRUE;                     // 标记本扫描周期允许刷新一次温控计算。
ELSE
    uiTempTickDiv := uiTempTickDiv + 1;         // 尚未达到 100ms 时继续累加 1ms 基础拍计数。
END_IF;

(* 先同步 HMI 参数边界，确保 HMI 下发的新工艺值先写入在线参数区。 *)
gvl_fbHMIParaInterface(
    stMachinePara := gvl_stPara,                // 传入机器在线工艺参数，供 HMI 接口执行读回与参数覆盖。
    stHMIPara := gvl_stHMIPara,                 // 传入 HMI 编辑缓冲区，供 HMI 页面维护配方编辑态。
    stCommand := gvl_stHMIParaCommand,          // 传入 HMI 参数同步命令，驱动读回、应用和脏标记清除。
    stMachineStatus := gvl_stStatus,            // 传入整机状态，便于 HMI 接口在机器忙碌时拦截参数下发。
    stStatus => gvl_stHMIParaStatus             // 回写 HMI 参数接口状态，供画面显示同步结果和拦截原因。
);

(* 再先调度顶层面板，把原始面板 IO 解码为按键结构，并把关键按键回灌到独立面板命令源。 *)
gvl_fbPanelDispatcher(
    stPanelButtons := gvl_stPanelButtons,       // 把全局综合面板按键边界交给面板调度块，统一回写键值和灯值。
    stPanelIO := gvl_stPanelIO,                 // 把全局面板原始 IO 边界交给面板调度块，统一处理输入解码与输出汇总。
    stCommandSource := gvl_stPanelCommandSource, // 把全局面板命令源边界交给面板调度块，让面板先只回灌自己的命令来源。
    ePanelModel := gvl_ePanelModel,             // 传入当前顶层选择的硬件面板型号，决定本拍调度哪个具体型号块。
    stStatus := gvl_stStatus,                   // 传入上一拍机器总状态，供面板调度块回写模式灯和动作灯。
    stSensor := gvl_stSensor                    // 传入现场传感器边界，供面板调度块回写马达/液压类状态灯。
);

(* 再把各命令源统一仲裁为最终机器命令，供顶层温控和机器主控共同消费。 *)
stBaseCommandSnapshot := gvl_stCommand;         // 先拍下当前扫描周期外部入口已经写入的基础机器命令，避免仲裁时直接覆盖掉公共控制字段。

gvl_fbCommandArbiter(
    stBaseCommandIn := stBaseCommandSnapshot,         // 把当前扫描周期的基础机器命令快照送入仲裁块，保留外部入口写入的公共控制字段。
    stPanelCommandSourceIn := gvl_stPanelCommandSource, // 把面板命令源送入顶层仲裁块，当前版本只用该源覆盖模式与手动字段。
    stCommandOut => gvl_stCommand                      // 回写仲裁后的最终机器命令，供后续顶层功能块统一消费。
);

(* 顶层独立处理温控系统，不再把温控结果并入机器主控。 *)
gvl_fbEK312(
    bStart := gvl_stCommand.stManual.bTempStart, // 直接把顶层温控启动命令送入温控块。
    bStop := gvl_stCommand.bStop,                // 机器停止时同步通知温控块退出执行态。
    bReset := gvl_stCommand.bReset,              // 机器复位时同步清空温控块内部状态。
    bLogicTick100msIn := bTempTick100ms,         // 把顶层 100ms 温控刷新拍送入温控块，让温控块每拍都被调用但只在该拍做一轮计算。
    bR0 := gvl_stCommand.stManual.bR0,           // 直接把第 0 组人工加热命令送入温控块。
    bR1 := gvl_stCommand.stManual.bR1,           // 直接把第 1 组人工加热命令送入温控块。
    bR2 := gvl_stCommand.stManual.bR2,           // 直接把第 2 组人工加热命令送入温控块。
    bR3 := gvl_stCommand.stManual.bR3,           // 直接把第 3 组人工加热命令送入温控块。
    stInPara := gvl_stPara.stEK312InPara,        // 把在线温控参数传给顶层温控块做 100ms 刷新计算。
    stOutPara => gvl_stTempOutPara               // 顶层直接回写温控输出结构，供 HMI 和其他顶层逻辑读取。
);

(* 再执行机器主控，由主控统一驱动模式管理、自动流程和全部执行模块。 *)
gvl_fbMachineController(
    stCommand := gvl_stCommand,                 // 传入机器公共命令，驱动模式路由、模块启动和复位逻辑。
    stPara := gvl_stPara,                       // 传入机器在线工艺参数，供主控分发给各子模块。
    stSensor := gvl_stSensor,                   // 传入现场输入与轴反馈，供主控和子模块做互锁判断。
    bLogicTick10msIn := bLogicTick10ms,         // 把顶层 10ms 工艺节拍送给主控，让主控只在该拍刷新模式路由和自动流程。
    stStatus => gvl_stStatus,                   // 回写机器级总状态，供 HMI 和上位调用链读取。
    stClampAxis => gvl_stClampAxis,             // 回写合模轴命令与反馈镜像，供后续轴控层或监控层读取。
    stMoldAdjustAxis => gvl_stMoldAdjustAxis,   // 回写调模轴命令与反馈镜像，供后续轴控层或监控层读取。
    stNozzleAxis => gvl_stNozzleAxis,           // 回写座台轴命令与反馈镜像，供后续轴控层或监控层读取。
    stInjectAxis => gvl_stInjectAxis,           // 回写射胶轴命令与反馈镜像，供后续轴控层或监控层读取。
    stMeterAxis => gvl_stMeterAxis,             // 回写储料轴命令与反馈镜像，供后续轴控层或监控层读取。
    stEjectAxis => gvl_stEjectAxis,             // 回写托模轴命令与反馈镜像，供后续轴控层或监控层读取。
    stCoreAxis => gvl_stCoreAxis,               // 回写中子轴命令与反馈镜像，供后续轴控层或监控层读取。
    aCoreAllow => gvl_aCoreAllow                // 回写合模允许中子动作数组，供其他联锁逻辑读取。
);
END_PROGRAM
